# B&R Automation Studio project CControl (part 3)

#### Main.st
```iecst
PROGRAM _INIT

END_PROGRAM

PROGRAM _CYCLIC

	//Zeitticks generieren
	fbLascoZdxx_0(IN 	:= Echtzeit.Sekunde);
	sekTick				:= fbLascoZdxx_0.Q;

	//Modul 2 bei Entfeuchter-Typen 7, 8, 9 und 10 (10 ist Reserve, eigene Einstellungen möglich)
	gModul2Vorhanden	:= (Betriebsparameter.Entfeuchter.IndexType = 7) OR (Betriebsparameter.Entfeuchter.IndexType = 8) OR (Betriebsparameter.Entfeuchter.IndexType = 9) OR
	(Betriebsparameter.Entfeuchter.IndexType = 10);

	//Ölsumpheizung Modul 1 **********************************************************************************************************************************************************************

	//Eingänge
	Aktoren.OelsumpfheizungModul1.EintrittTemp					:= aiEintrittTemperatur;
	Aktoren.OelsumpfheizungModul1.StatusSensorEintrittOk		:= NOT alarmFehler[FEHLER_SENSOR_EINTRITT];

	//GUI-Parameter
	Aktoren.OelsumpfheizungModul1.parTempOelsumpfheizungEin		:= 0.0;
	Aktoren.OelsumpfheizungModul1.parTempOelsumpfheizungAus		:= 0.0;

	//Ausgänge
	doOelsumpfheizungEinModul1									:= Aktoren.OelsumpfheizungModul1.OelsumpfheizungEin;

	//Status
	IF  doOelsumpfheizungEinModul1 THEN
		gStatusAnlage.Aktor[AKTOR_OELSUMPFHEIZUNG_MOD1]	:= STATUS_AKTIV;
	ELSE
		gStatusAnlage.Aktor[AKTOR_OELSUMPFHEIZUNG_MOD1]	:= STATUS_NICHT_AKTIV;
	END_IF

	//Ölsumpheizung Modul 2 **********************************************************************************************************************************************************************

	//Eingänge
	Aktoren.OelsumpfheizungModul2.EintrittTemp					:= aiEintrittTemperatur;
	Aktoren.OelsumpfheizungModul2.StatusSensorEintrittOk		:= NOT alarmFehler[FEHLER_SENSOR_EINTRITT];

	//GUI-Parameter
	Aktoren.OelsumpfheizungModul2.parTempOelsumpfheizungEin		:= 0.0;
	Aktoren.OelsumpfheizungModul2.parTempOelsumpfheizungAus		:= 0.0;

	//Ausgänge
	doOelsumpfheizungEinModul2										:= Aktoren.OelsumpfheizungModul2.OelsumpfheizungEin;

	//Status
	IF  doOelsumpfheizungEinModul2 THEN
		gStatusAnlage.Aktor[AKTOR_OELSUMPFHEIZUNG_MOD2]	:= STATUS_AKTIV;
	ELSE
		gStatusAnlage.Aktor[AKTOR_OELSUMPFHEIZUNG_MOD2]	:= STATUS_NICHT_AKTIV;
	END_IF

	//Kompressor Modul 1 **********************************************************************************************************************************************************************

	//Eingänge
	Aktoren.KompressorModul1.EintrittFeuchte			:= aiEintrittFeuchte;
	Aktoren.KompressorModul1.Niederdruck				:= aiNiederdruckModul1;
	Aktoren.KompressorModul1.Hochdruck					:= aiHochdruckModul1;
	Aktoren.KompressorModul1.KlappenumschaltungAkiv		:= Aktoren.VentUndKlappen.UmschaltungAktiv OR Strombegrenzung.StrombegrenzungEin OR
	(diDrehzahlbegrVentilator1 AND Boxen.EntfeuchterVonVent1Abhaengig) OR (diDrehzahlbegrVentilator2 AND Boxen.EntfeuchterVonVent2Abhaengig);
	Aktoren.KompressorModul1.BetriebsmldgVentilator		:= (doVentilator1Ein AND Boxen.EntfeuchterVonVent1Abhaengig) OR
	(doVentilator2Ein AND Boxen.EntfeuchterVonVent2Abhaengig) OR (diVentilator1InBetrieb AND Boxen.EntfeuchterInselbetrieb);
	Aktoren.KompressorModul1.BetriebsmldgKompressor		:= diBetriebsmldgKompressorModul1;
	Aktoren.KompressorModul1.StatusSensorEintrittOk		:= NOT alarmFehler[FEHLER_SENSOR_EINTRITT];
	Aktoren.KompressorModul1.StatusSensorNiederdruckOk	:= NOT alarmFehler[FEHLER_SENSOR_NIEDERDRUCK_MOD1];
	Aktoren.KompressorModul1.diHochdruckOk				:= diHochdruckOkModul1;
	Aktoren.KompressorModul1.diNiederdruckOk			:= diNiederdruckOkModul1;
	Aktoren.KompressorModul1.SicherheitOk				:= NOT alarmFehler[FEHLER_HOCHDRUCK_MODUL1] AND NOT alarmFehler[FEHLER_NIEDERDRUCK_MODUL1] AND NOT alarmFehler[FEHLER_VOLLSCHUTZ_KOMPR_MOD1] AND NOT
	alarmFehler[FEHLER_OELDRUCK_KOMPR_MOD1] AND NOT alarmFehler[FEHLER_EINTRITT_TEMP_ZU_HOCH] AND NOT alarmFehler[FEHLER_EINTRITT_TEMP_ZU_NIEDRIG];

	//GUI-Parameter
	Aktoren.KompressorModul1.QuitFehler						:= hmiButtons.QuitFehler;
	Aktoren.KompressorModul1.parEinschaltverzAbtau			:= Betriebsparameter.Entfeuchter.EinschaltverzAbtau;
	Aktoren.KompressorModul1.parAusschaltverzAbtau			:= Betriebsparameter.Entfeuchter.AusschaltverzAbtau;
	Aktoren.KompressorModul1.parEinschaltverzKompressor		:= Betriebsparameter.Entfeuchter.EinschaltverzKompressor;
	Aktoren.KompressorModul1.parEinschaltverzMagnetventil	:= Betriebsparameter.Kompressor1.EinschaltverzMagnetventil;
	Aktoren.KompressorModul1.parFeuchteEin					:= Betriebsparameter.Entfeuchter.EintrittFeuchteEin;
	Aktoren.KompressorModul1.parFeuchteAus					:= Betriebsparameter.Entfeuchter.EintrittFeuchteAus;
	Aktoren.KompressorModul1.parNiederdruckMin				:= Betriebsparameter.Kompressor1.NiederdruckMin;
	Aktoren.KompressorModul1.parNiederdruckMax				:= Betriebsparameter.Kompressor1.NiederdruckMax;
	Aktoren.KompressorModul1.parNiederdruckPumpdown			:= Betriebsparameter.Kompressor1.NiederdruckPumpDown;
	Aktoren.KompressorModul1.parHochdruckMax				:= Betriebsparameter.Kompressor1.HochdruckMax;
	Aktoren.KompressorModul1.parVerzStandbyBeiKlappenumsch	:= Betriebsparameter.Entfeuchter.VerzStandbyHochdruckMax;
	Aktoren.KompressorModul1.DrehzahlMin					:= Betriebsparameter.Kompressor1.DrehzahlMin;
	Aktoren.KompressorModul1.DrehzahlMax					:= Betriebsparameter.Kompressor1.DrehzahlMax;
	Aktoren.KompressorModul1.RampeUp						:= Betriebsparameter.Kompressor1.RampeUp;
	Aktoren.KompressorModul1.RampeDown						:= Betriebsparameter.Kompressor1.RampeDown;

	//Ausgänge
	doKompressorEinModul1									:= Aktoren.KompressorModul1.FreigabeKompressorOut AND diHochdruckOkModul1 AND diNiederdruckOkModul1;
	aoDrehzahlvorgKompressorModul1							:= Aktoren.KompressorModul1.DrehzahlOut;
	doMagnetventilEinModul1									:= Aktoren.KompressorModul1.MagnetventilOut;

	//Status
	IF doKompressorEinModul1 THEN
		gStatusAnlage.Aktor[AKTOR_KOMPRESSOR_MOD1]			:= STATUS_AKTIV;
	ELSIF Aktoren.KompressorModul1.StoerungOut THEN
		gStatusAnlage.Aktor[AKTOR_KOMPRESSOR_MOD1]			:= STATUS_STOERUNG;
	ELSIF (Aktoren.KompressorModul1.Automatik OR Aktoren.KompressorModul1.Dauerbetrieb) AND Boxen.FreigabeLuftentfeuchter AND NOT doKompressorEinModul1 THEN
		gStatusAnlage.Aktor[AKTOR_KOMPRESSOR_MOD1]			:= STATUS_ENTF_STANDBY;
	ELSIF Aktoren.KompressorModul1.AbtauungAktiv THEN
		gStatusAnlage.Aktor[AKTOR_KOMPRESSOR_MOD1]			:= STATUS_ENTF_ABTAUUNG;
	ELSE
		gStatusAnlage.Aktor[AKTOR_KOMPRESSOR_MOD1]			:= STATUS_NICHT_AKTIV;
	END_IF

	//Status
	IF  doMagnetventilEinModul1 THEN
		gStatusAnlage.Aktor[AKTOR_MAGNETVENTIL_MOD1]		:= STATUS_AKTIV;
	ELSE
		gStatusAnlage.Aktor[AKTOR_MAGNETVENTIL_MOD1]		:= STATUS_NICHT_AKTIV;
	END_IF

	//Kompressor Modul 2 **********************************************************************************************************************************************************************

	//Eingänge
	Aktoren.KompressorModul2.EintrittFeuchte			:= aiEintrittFeuchte;
	Aktoren.KompressorModul2.Niederdruck				:= aiNiederdruckModul2;
	Aktoren.KompressorModul2.Hochdruck					:= aiHochdruckModul2;
	Aktoren.KompressorModul2.KlappenumschaltungAkiv		:= Aktoren.VentUndKlappen.UmschaltungAktiv OR Strombegrenzung.StrombegrenzungEin OR
	(diDrehzahlbegrVentilator1 AND Boxen.EntfeuchterVonVent1Abhaengig) OR (diDrehzahlbegrVentilator2 AND Boxen.EntfeuchterVonVent2Abhaengig);
	Aktoren.KompressorModul2.BetriebsmldgVentilator		:= (doVentilator1Ein AND Boxen.EntfeuchterVonVent1Abhaengig) OR
	(doVentilator2Ein AND Boxen.EntfeuchterVonVent2Abhaengig) OR (diVentilator1InBetrieb AND Boxen.EntfeuchterInselbetrieb);
	Aktoren.KompressorModul2.BetriebsmldgKompressor		:= diBetriebsmldgKompressorModul2;
	Aktoren.KompressorModul2.StatusSensorEintrittOk		:= NOT alarmFehler[FEHLER_SENSOR_EINTRITT];
	Aktoren.KompressorModul2.StatusSensorNiederdruckOk	:= NOT alarmFehler[FEHLER_SENSOR_NIEDERDRUCK_MOD2];
	Aktoren.KompressorModul2.diHochdruckOk				:= diHochdruckOkModul2;
	Aktoren.KompressorModul2.diNiederdruckOk			:= diNiederdruckOkModul2;
	Aktoren.KompressorModul2.SicherheitOk				:= NOT alarmFehler[FEHLER_HOCHDRUCK_MODUL2] AND NOT alarmFehler[FEHLER_NIEDERDRUCK_MODUL2] AND NOT alarmFehler[FEHLER_VOLLSCHUTZ_KOMPR_MOD2] AND NOT
	alarmFehler[FEHLER_OELDRUCK_KOMPR_MOD2] AND NOT alarmFehler[FEHLER_EINTRITT_TEMP_ZU_HOCH] AND NOT alarmFehler[FEHLER_EINTRITT_TEMP_ZU_NIEDRIG];

	//GUI-Parameter
	Aktoren.KompressorModul2.QuitFehler						:= hmiButtons.QuitFehler;
	Aktoren.KompressorModul2.parEinschaltverzAbtau			:= Betriebsparameter.Entfeuchter.EinschaltverzAbtau;
	Aktoren.KompressorModul2.parAusschaltverzAbtau			:= Betriebsparameter.Entfeuchter.AusschaltverzAbtau;
	Aktoren.KompressorModul2.parEinschaltverzKompressor		:= Betriebsparameter.Entfeuchter.EinschaltverzKompressor + Betriebsparameter.Entfeuchter.AnlaufverzModul2;
	Aktoren.KompressorModul2.parEinschaltverzMagnetventil	:= Betriebsparameter.Kompressor1.EinschaltverzMagnetventil;
	Aktoren.KompressorModul2.parFeuchteEin					:= Betriebsparameter.Entfeuchter.EintrittFeuchteEin;
	Aktoren.KompressorModul2.parFeuchteAus					:= Betriebsparameter.Entfeuchter.EintrittFeuchteAus;
	Aktoren.KompressorModul2.parNiederdruckMin				:= Betriebsparameter.Kompressor1.NiederdruckMin;
	Aktoren.KompressorModul2.parNiederdruckMax				:= Betriebsparameter.Kompressor1.NiederdruckMax;
	Aktoren.KompressorModul2.parNiederdruckPumpdown			:= Betriebsparameter.Kompressor1.NiederdruckPumpDown;
	Aktoren.KompressorModul2.parHochdruckMax				:= Betriebsparameter.Kompressor1.HochdruckMax;
	Aktoren.KompressorModul2.parVerzStandbyBeiKlappenumsch	:= Betriebsparameter.Entfeuchter.VerzStandbyHochdruckMax;
	Aktoren.KompressorModul2.DrehzahlMin					:= Betriebsparameter.Kompressor2.DrehzahlMin;
	Aktoren.KompressorModul2.DrehzahlMax					:= Betriebsparameter.Kompressor2.DrehzahlMax;
	Aktoren.KompressorModul2.RampeUp						:= Betriebsparameter.Kompressor2.RampeUp;
	Aktoren.KompressorModul2.RampeDown						:= Betriebsparameter.Kompressor2.RampeDown;

	//Ausgänge
	doKompressorEinModul2									:= Aktoren.KompressorModul2.FreigabeKompressorOut AND diHochdruckOkModul2 AND diNiederdruckOkModul2;
	aoDrehzahlvorgKompressorModul2							:= Aktoren.KompressorModul2.DrehzahlOut;
	doMagnetventilEinModul2									:= Aktoren.KompressorModul2.MagnetventilOut;

	//Status
	IF doKompressorEinModul2 THEN
		gStatusAnlage.Aktor[AKTOR_KOMPRESSOR_MOD2]			:= STATUS_AKTIV;
	ELSIF Aktoren.KompressorModul2.StoerungOut THEN
		gStatusAnlage.Aktor[AKTOR_KOMPRESSOR_MOD2]			:= STATUS_STOERUNG;
	ELSIF (Aktoren.KompressorModul2.Automatik OR Aktoren.KompressorModul2.Dauerbetrieb) AND Boxen.FreigabeLuftentfeuchter AND NOT doKompressorEinModul2 THEN
		gStatusAnlage.Aktor[AKTOR_KOMPRESSOR_MOD2]			:= STATUS_ENTF_STANDBY;
	ELSIF Aktoren.KompressorModul2.AbtauungAktiv THEN
		gStatusAnlage.Aktor[AKTOR_KOMPRESSOR_MOD2]			:= STATUS_ENTF_ABTAUUNG;
	ELSE
		gStatusAnlage.Aktor[AKTOR_KOMPRESSOR_MOD2]			:= STATUS_NICHT_AKTIV;
	END_IF

	//Status
	IF  doMagnetventilEinModul2 THEN
		gStatusAnlage.Aktor[AKTOR_MAGNETVENTIL_MOD2]		:= STATUS_AKTIV;
	ELSE
		gStatusAnlage.Aktor[AKTOR_MAGNETVENTIL_MOD2]		:= STATUS_NICHT_AKTIV;
	END_IF

	//Entfeuchter Fremdgerät **********************************************************************************************************************************************************************

	//Eingänge
	Aktoren.EntfeuchterFremd.BetriebsmldgEntfeuchter	:= diEntfeuchterFremdInBetrieb;
	Aktoren.EntfeuchterFremd.BetriebsmldgVentilator		:= diVentilator1InBetrieb;

	Aktoren.EntfeuchterFremd.WitterungIstSchlecht		:= (fbSchlechtwetterBox1.WetterIstSchlecht AND Betriebsparameter.Boxen[1].Luftentfeuchter AND Boxen.Box1Out.BoxAktiv) OR
	(fbSchlechtwetterBox2.WetterIstSchlecht AND Betriebsparameter.Boxen[2].Luftentfeuchter AND Boxen.Box2Out.BoxAktiv) OR
	(fbSchlechtwetterBox3.WetterIstSchlecht AND Betriebsparameter.Boxen[3].Luftentfeuchter AND Boxen.Box3Out.BoxAktiv) OR
	(fbSchlechtwetterBox4.WetterIstSchlecht AND Betriebsparameter.Boxen[4].Luftentfeuchter AND Boxen.Box4Out.BoxAktiv) OR
	(fbSchlechtwetterBox5.WetterIstSchlecht AND Betriebsparameter.Boxen[5].Luftentfeuchter AND Boxen.Box5Out.BoxAktiv) OR
	(fbSchlechtwetterBox6.WetterIstSchlecht AND Betriebsparameter.Boxen[6].Luftentfeuchter AND Boxen.Box6Out.BoxAktiv);
	Aktoren.EntfeuchterFremd.StoerungIn					:= diEntfeuchterFremdStoerung;

	//GUI-Parameter
	Aktoren.EntfeuchterFremd.parEinschaltverzKompressor	:= Betriebsparameter.Entfeuchter.EinschaltverzKompressor;
	Aktoren.EntfeuchterFremd.parVerzBetriebEntfeuchter	:= Betriebsparameter.Entfeuchter.VerzBetriebsmeldung;
	Aktoren.EntfeuchterFremd.parVerzStoerung			:= REAL_TO_UDINT(Betriebsparameter.Allgemein.VerzoegerungFehler * 1000);
	Aktoren.EntfeuchterFremd.QuitFehler					:= hmiButtons.QuitFehler;

	//Ausgänge
	doEntfFremdFreigabe									:= Aktoren.EntfeuchterFremd.FreigabeKompressorOut;

	//Status
	IF doEntfFremdFreigabe THEN
		IF diEntfeuchterFremdInBetrieb THEN
			gStatusAnlage.Aktor[AKTOR_ENTFEUCHTER_FREMD]		:= STATUS_AKTIV;
		ELSE
			gStatusAnlage.Aktor[AKTOR_ENTFEUCHTER_FREMD]		:= STATUS_ENTF_STANDBY;
		END_IF
	ELSIF Aktoren.EntfeuchterFremd.StoerungOut THEN
		gStatusAnlage.Aktor[AKTOR_ENTFEUCHTER_FREMD]		:= STATUS_STOERUNG;
	ELSE
		gStatusAnlage.Aktor[AKTOR_ENTFEUCHTER_FREMD]		:= STATUS_NICHT_AKTIV;
	END_IF

	//Abluftklappe **********************************************************************************************************************************************************************

	//Eingänge
	Aktoren.Abluftklappe.AbluftFeuchteIst			:= aiAbluftFeuchte;
	Aktoren.Abluftklappe.EndlageOffen				:= diAbluftklappeOffen;
	Aktoren.Abluftklappe.EndlageGeschl				:= diAbluftklappeGeschl;

	//GUI-Parameter
	Aktoren.Abluftklappe.AbluftFeuchteSoll			:= Betriebsparameter.Abluftklappe.AbluftfeuchteMax;
	Aktoren.Abluftklappe.Hysterese					:= Betriebsparameter.Abluftklappe.Hysterese;
	Aktoren.Abluftklappe.Laufzeit					:= Betriebsparameter.Abluftklappe.Laufzeit;
	Aktoren.Abluftklappe.Quit						:= hmiButtons.QuitFehler;

	//Ausgänge
	doAbluftklappeFreigabe							:= Aktoren.Abluftklappe.OeffnenOut AND NOT Aktoren.Abluftklappe.SchliessenOut;
	doAbluftklappeOeffnen							:= Aktoren.Abluftklappe.OeffnenOut;
	doAbluftklappeSchliessen						:= Aktoren.Abluftklappe.SchliessenOut;

	//Status
	IF doAbluftklappeFreigabe AND NOT diAbluftklappeOffen AND (Betriebsparameter.Abluftklappe.Laufzeit <> 0) THEN
		gStatusAnlage.Aktor[AKTOR_ABLUFTKLAPPE]			:= STATUS_AKTIV;
	ELSIF (NOT doAbluftklappeFreigabe) AND NOT diAbluftklappeGeschl AND (Betriebsparameter.Abluftklappe.Laufzeit <> 0) THEN
		gStatusAnlage.Aktor[AKTOR_ABLUFTKLAPPE]			:= STATUS_AKTIV;
	ELSIF Aktoren.Abluftklappe.FehlerLaufzeit THEN
		gStatusAnlage.Aktor[AKTOR_ABLUFTKLAPPE]			:= STATUS_STOERUNG;
	ELSIF doAbluftklappeFreigabe AND (diAbluftklappeOffen OR (Betriebsparameter.Abluftklappe.Laufzeit = 0)) THEN
		gStatusAnlage.Aktor[AKTOR_ABLUFTKLAPPE]			:= STATUS_OFFEN;
	ELSIF (NOT doAbluftklappeFreigabe) AND (diAbluftklappeGeschl OR (Betriebsparameter.Abluftklappe.Laufzeit = 0)) THEN
		gStatusAnlage.Aktor[AKTOR_ABLUFTKLAPPE]			:= STATUS_GESCHLOSSEN;
	ELSE
		gStatusAnlage.Aktor[AKTOR_ABLUFTKLAPPE]			:= STATUS_NICHT_AKTIV;
	END_IF

	//Abluftventilator **********************************************************************************************************************************************************************

	//Eingänge
	Aktoren.Abluftventilator.AbluftFeuchteIst		:= aiAbluftFeuchte;
	Aktoren.Abluftventilator.VentilatorInBetrieb	:= diAbluftventInBetrieb;
	Aktoren.Abluftventilator.RampeUp				:= 10;
	Aktoren.Abluftventilator.RampeDown				:= 10;

	//GUI-Parameter
	Aktoren.Abluftventilator.DrehzahlMin			:= Betriebsparameter.Abluftventilator.DrehzahlMin;
	Aktoren.Abluftventilator.DrehzahlMax			:= Betriebsparameter.Abluftventilator.DrehzahlMax;
	Aktoren.Abluftventilator.AbluftFeuchteSoll		:= Betriebsparameter.Abluftventilator.AbluftfeuchteMax;
	Aktoren.Abluftventilator.Hysterese				:= Betriebsparameter.Abluftventilator.Hysterese;
	Aktoren.Abluftventilator.QuitFehler				:= hmiButtons.QuitFehler;

	//Ausgänge
	doAbluftventilatorEin							:= Aktoren.Abluftventilator.FreigabeVentilatorOut;
	aoDrehzahlvorgAbluftventilator					:= Aktoren.Abluftventilator.DrehzahlVentilatorOut;

	//Status
	IF doAbluftventilatorEin THEN
		gStatusAnlage.Aktor[AKTOR_ABLUFTVENTILATOR]		:= STATUS_AKTIV;
	ELSIF Aktoren.Abluftventilator.FehlerOut THEN
		gStatusAnlage.Aktor[AKTOR_ABLUFTVENTILATOR]		:= STATUS_STOERUNG;
	ELSE
		gStatusAnlage.Aktor[AKTOR_ABLUFTVENTILATOR]		:= STATUS_NICHT_AKTIV;
	END_IF

	//Ventilatoren, Bypassklappe, Umschaltklappen und Klappen für Boxen **********************************************************************************************************************

	//Eingänge
	Aktoren.VentUndKlappen.Freigabe						:= TRUE;
	Aktoren.VentUndKlappen.BypassklVonVent1Abhaengig	:= Boxen.BypassklVonVent1Abhaengig;
	Aktoren.VentUndKlappen.BypassklVonVent2Abhaengig	:= Boxen.BypassklVonVent2Abhaengig;
	Aktoren.VentUndKlappen.Boxenkl1VonVent1Abhaengig	:= Boxen.Boxenkl1VonVent1Abhaengig;
	Aktoren.VentUndKlappen.Boxenkl2VonVent1Abhaengig	:= Boxen.Boxenkl2VonVent1Abhaengig;
	Aktoren.VentUndKlappen.Boxenkl3VonVent1Abhaengig	:= Boxen.Boxenkl3VonVent1Abhaengig;
	Aktoren.VentUndKlappen.Boxenkl4VonVent1Abhaengig	:= Boxen.Boxenkl4VonVent1Abhaengig;
	Aktoren.VentUndKlappen.Boxenkl5VonVent1Abhaengig	:= Boxen.Boxenkl5VonVent1Abhaengig;
	Aktoren.VentUndKlappen.Boxenkl6VonVent1Abhaengig	:= Boxen.Boxenkl6VonVent1Abhaengig;
	Aktoren.VentUndKlappen.Boxenkl1VonVent2Abhaengig	:= Boxen.Boxenkl1VonVent2Abhaengig;
	Aktoren.VentUndKlappen.Boxenkl2VonVent2Abhaengig	:= Boxen.Boxenkl2VonVent2Abhaengig;
	Aktoren.VentUndKlappen.Boxenkl3VonVent2Abhaengig	:= Boxen.Boxenkl3VonVent2Abhaengig;
	Aktoren.VentUndKlappen.Boxenkl4VonVent2Abhaengig	:= Boxen.Boxenkl4VonVent2Abhaengig;
	Aktoren.VentUndKlappen.Boxenkl5VonVent2Abhaengig	:= Boxen.Boxenkl5VonVent2Abhaengig;
	Aktoren.VentUndKlappen.Boxenkl6VonVent2Abhaengig	:= Boxen.Boxenkl6VonVent2Abhaengig;
	Aktoren.VentUndKlappen.UmluftklVonVent1Abhaengig	:= Betriebsparameter.Ausstattung.Vent1AusWennUmschUmluftkl;
	Aktoren.VentUndKlappen.UmluftklVonVent2Abhaengig	:= Betriebsparameter.Ausstattung.Vent2AusWennUmschUmluftkl;
	Aktoren.VentUndKlappen.EndlBoxenklappe1Geschl		:= diBox1Geschl;
	Aktoren.VentUndKlappen.EndlBoxenklappe1Offen		:= diBox1Offen;
	Aktoren.VentUndKlappen.EndlBoxenklappe2Geschl		:= diBox2Geschl;
	Aktoren.VentUndKlappen.EndlBoxenklappe2Offen		:= diBox2Offen;
	Aktoren.VentUndKlappen.EndlBoxenklappe3Geschl		:= diBox3Geschl;
	Aktoren.VentUndKlappen.EndlBoxenklappe3Offen		:= diBox3Offen;
	Aktoren.VentUndKlappen.EndlBoxenklappe4Geschl		:= diBox4Geschl;
	Aktoren.VentUndKlappen.EndlBoxenklappe4Offen		:= diBox4Offen;
	Aktoren.VentUndKlappen.EndlBoxenklappe5Geschl		:= diBox5Geschl;
	Aktoren.VentUndKlappen.EndlBoxenklappe5Offen		:= diBox5Offen;
	Aktoren.VentUndKlappen.EndlBoxenklappe6Geschl		:= diBox6Geschl;
	Aktoren.VentUndKlappen.EndlBoxenklappe6Offen		:= diBox6Offen;
	Aktoren.VentUndKlappen.EndlBypassGeschl				:= diBypassklappeGeschl;
	Aktoren.VentUndKlappen.EndlBypassOffen				:= diBypassklappeOffen;
	Aktoren.VentUndKlappen.EndlBypassGeschl				:= diBypassklappeGeschl;
	Aktoren.VentUndKlappen.EndlBypassOffen				:= diBypassklappeOffen;
	Aktoren.VentUndKlappen.EndlUmschaltkl1Geschl		:= diUmschaltklappe1Geschl;
	Aktoren.VentUndKlappen.EndlUmschaltkl1Offen			:= diUmschaltklappe1Offen;
	Aktoren.VentUndKlappen.EndlUmschaltkl2Geschl		:= diUmschaltklappe2Geschl;
	Aktoren.VentUndKlappen.EndlUmschaltkl2Offen			:= diUmschaltklappe2Offen;
	Aktoren.VentUndKlappen.LuftaufbereitungInBetrieb	:= doKompressorEinModul1 OR doKompressorEinModul2 OR Aktoren.Warmluftofen.WarmluftofenAktiv OR
	Aktoren.Scheitholzofen.ScheitholzofenAktiv OR doHeizregisterEin;
	Aktoren.VentUndKlappen.Ventilator1InBetrieb			:= diVentilator1InBetrieb;
	Aktoren.VentUndKlappen.Ventilator2InBetrieb			:= diVentilator2InBetrieb;
	Aktoren.VentUndKlappen.Boxenklappe1Vorhanden		:= (Betriebsparameter.Boxen[1].StellungKlappe1 <> FBBOX_NICHT_VERWENDET) OR
	(Betriebsparameter.Boxen[2].StellungKlappe1 <> FBBOX_NICHT_VERWENDET) OR (Betriebsparameter.Boxen[3].StellungKlappe1 <> FBBOX_NICHT_VERWENDET) OR
	(Betriebsparameter.Boxen[4].StellungKlappe1 <> FBBOX_NICHT_VERWENDET) OR (Betriebsparameter.Boxen[5].StellungKlappe1 <> FBBOX_NICHT_VERWENDET) OR
	(Betriebsparameter.Boxen[6].StellungKlappe1 <> FBBOX_NICHT_VERWENDET);
	Aktoren.VentUndKlappen.Boxenklappe2Vorhanden		:= (Betriebsparameter.Boxen[1].StellungKlappe2 <> FBBOX_NICHT_VERWENDET) OR
	(Betriebsparameter.Boxen[2].StellungKlappe2 <> FBBOX_NICHT_VERWENDET) OR (Betriebsparameter.Boxen[3].StellungKlappe2 <> FBBOX_NICHT_VERWENDET) OR
	(Betriebsparameter.Boxen[4].StellungKlappe2 <> FBBOX_NICHT_VERWENDET) OR (Betriebsparameter.Boxen[5].StellungKlappe2 <> FBBOX_NICHT_VERWENDET) OR
	(Betriebsparameter.Boxen[6].StellungKlappe2 <> FBBOX_NICHT_VERWENDET);
	Aktoren.VentUndKlappen.Boxenklappe3Vorhanden		:= (Betriebsparameter.Boxen[1].StellungKlappe3 <> FBBOX_NICHT_VERWENDET) OR
	(Betriebsparameter.Boxen[2].StellungKlappe3 <> FBBOX_NICHT_VERWENDET) OR (Betriebsparameter.Boxen[3].StellungKlappe3 <> FBBOX_NICHT_VERWENDET) OR
	(Betriebsparameter.Boxen[4].StellungKlappe3 <> FBBOX_NICHT_VERWENDET) OR (Betriebsparameter.Boxen[5].StellungKlappe3 <> FBBOX_NICHT_VERWENDET) OR
	(Betriebsparameter.Boxen[6].StellungKlappe3 <> FBBOX_NICHT_VERWENDET);
	Aktoren.VentUndKlappen.Boxenklappe4Vorhanden		:= (Betriebsparameter.Boxen[1].StellungKlappe4 <> FBBOX_NICHT_VERWENDET) OR
	(Betriebsparameter.Boxen[2].StellungKlappe4 <> FBBOX_NICHT_VERWENDET) OR (Betriebsparameter.Boxen[3].StellungKlappe4 <> FBBOX_NICHT_VERWENDET) OR
	(Betriebsparameter.Boxen[4].StellungKlappe4 <> FBBOX_NICHT_VERWENDET) OR (Betriebsparameter.Boxen[5].StellungKlappe4 <> FBBOX_NICHT_VERWENDET) OR
	(Betriebsparameter.Boxen[6].StellungKlappe4 <> FBBOX_NICHT_VERWENDET);
	Aktoren.VentUndKlappen.Boxenklappe5Vorhanden		:= (Betriebsparameter.Boxen[1].StellungKlappe5 <> FBBOX_NICHT_VERWENDET) OR
	(Betriebsparameter.Boxen[2].StellungKlappe5 <> FBBOX_NICHT_VERWENDET) OR (Betriebsparameter.Boxen[3].StellungKlappe5 <> FBBOX_NICHT_VERWENDET) OR
	(Betriebsparameter.Boxen[4].StellungKlappe5 <> FBBOX_NICHT_VERWENDET) OR (Betriebsparameter.Boxen[5].StellungKlappe5 <> FBBOX_NICHT_VERWENDET) OR
	(Betriebsparameter.Boxen[6].StellungKlappe5 <> FBBOX_NICHT_VERWENDET);
	Aktoren.VentUndKlappen.Boxenklappe6Vorhanden		:= (Betriebsparameter.Boxen[1].StellungKlappe6 <> FBBOX_NICHT_VERWENDET) OR
	(Betriebsparameter.Boxen[2].StellungKlappe6 <> FBBOX_NICHT_VERWENDET) OR (Betriebsparameter.Boxen[3].StellungKlappe6 <> FBBOX_NICHT_VERWENDET) OR
	(Betriebsparameter.Boxen[4].StellungKlappe6 <> FBBOX_NICHT_VERWENDET) OR (Betriebsparameter.Boxen[5].StellungKlappe6 <> FBBOX_NICHT_VERWENDET) OR
	(Betriebsparameter.Boxen[6].StellungKlappe6 <> FBBOX_NICHT_VERWENDET);

	//GUI-Parameter
	Aktoren.VentUndKlappen.QuitFehler					:= hmiButtons.QuitFehler;
	Aktoren.VentUndKlappen.AnlaufverzZweiterVent		:= Betriebsparameter.Schrittkette.AnlaufverzZweiterVentilator;
	Aktoren.VentUndKlappen.DrehzahlVent1Min				:= Betriebsparameter.Ventilator1.DrehzahlMin;
	Aktoren.VentUndKlappen.DrehzahlVent1Max				:= Betriebsparameter.Ventilator1.DrehzahlMax;
	Aktoren.VentUndKlappen.RampeVent1Up					:= Betriebsparameter.Ventilator1.ZeitRampeUp;
	Aktoren.VentUndKlappen.RampeVent1Down				:= Betriebsparameter.Ventilator1.ZeitRampeDown;
	Aktoren.VentUndKlappen.DrehzahlVent1Umsch			:= Betriebsparameter.Ventilator1.DrzUmschaltung;
	Aktoren.VentUndKlappen.DrzVent1UmschMitLuftaufb		:= Betriebsparameter.Ventilator1.DrzUmschaltungMitLuftaufb;
	Aktoren.VentUndKlappen.DrehzahlVent2Min				:= Betriebsparameter.Ventilator2.DrehzahlMin;
	Aktoren.VentUndKlappen.DrehzahlVent2Max				:= Betriebsparameter.Ventilator2.DrehzahlMax;
	Aktoren.VentUndKlappen.RampeVent2Up					:= Betriebsparameter.Ventilator2.ZeitRampeUp;
	Aktoren.VentUndKlappen.RampeVent2Down				:= Betriebsparameter.Ventilator2.ZeitRampeDown;
	Aktoren.VentUndKlappen.DrehzahlVent2Umsch			:= Betriebsparameter.Ventilator2.DrzUmschaltung;
	Aktoren.VentUndKlappen.DrzVent2UmschMitLuftaufb		:= Betriebsparameter.Ventilator2.DrzUmschaltungMitLuftaufb;
	Aktoren.VentUndKlappen.LaufzeitBypassklappe			:= Betriebsparameter.Bypassklappe.Laufzeit;
	Aktoren.VentUndKlappen.LaufzeitBoxenklappe1			:= Betriebsparameter.KlappenBoxen[1].Laufzeit;
	Aktoren.VentUndKlappen.LaufzeitBoxenklappe2			:= Betriebsparameter.KlappenBoxen[2].Laufzeit;
	Aktoren.VentUndKlappen.LaufzeitBoxenklappe3			:= Betriebsparameter.KlappenBoxen[3].Laufzeit;
	Aktoren.VentUndKlappen.LaufzeitBoxenklappe4			:= Betriebsparameter.KlappenBoxen[4].Laufzeit;
	Aktoren.VentUndKlappen.LaufzeitBoxenklappe5			:= Betriebsparameter.KlappenBoxen[5].Laufzeit;
	Aktoren.VentUndKlappen.LaufzeitBoxenklappe6			:= Betriebsparameter.KlappenBoxen[6].Laufzeit;
	Aktoren.VentUndKlappen.LaufzeitUmschaltklappe1		:= Betriebsparameter.Umschaltklappen.LaufzeitKlappe1;
	Aktoren.VentUndKlappen.LaufzeitUmschaltklappe2		:= Betriebsparameter.Umschaltklappen.LaufzeitKlappe2;
	Aktoren.VentUndKlappen.EndlagenVhdBoxenklappe1		:= Betriebsparameter.Ausstattung.EndlagenVhdBoxenklappe1;
	Aktoren.VentUndKlappen.EndlagenVhdBoxenklappe2		:= Betriebsparameter.Ausstattung.EndlagenVhdBoxenklappe2;
	Aktoren.VentUndKlappen.EndlagenVhdBoxenklappe3		:= Betriebsparameter.Ausstattung.EndlagenVhdBoxenklappe3;
	Aktoren.VentUndKlappen.EndlagenVhdBoxenklappe4		:= Betriebsparameter.Ausstattung.EndlagenVhdBoxenklappe4;
	Aktoren.VentUndKlappen.EndlagenVhdBoxenklappe5		:= Betriebsparameter.Ausstattung.EndlagenVhdBoxenklappe5;
	Aktoren.VentUndKlappen.EndlagenVhdBoxenklappe6		:= Betriebsparameter.Ausstattung.EndlagenVhdBoxenklappe6;
	Aktoren.VentUndKlappen.EndlagenVhdUmschaltklappe1	:= Betriebsparameter.Ausstattung.EndlagenVhdUmschaltklappe1;
	Aktoren.VentUndKlappen.EndlagenVhdUmschaltklappe2	:= Betriebsparameter.Ausstattung.EndlagenVhdUmschaltklappe1;//Option Endlagen Umschaltklappen nur für beide Klappen gleich einstellbar
	Aktoren.VentUndKlappen.EndlagenVhdBypassklappe		:= Betriebsparameter.Ausstattung.EndlagenVhdBypassklappe;

	//Ausgänge
	doVentilator1Ein									:= Aktoren.VentUndKlappen.FreigabeVentilator1Out;
	doVentilator2Ein									:= Aktoren.VentUndKlappen.FreigabeVentilator2Out;
	aoDrehzahlvorgVentilator1							:= Aktoren.VentUndKlappen.DrehzahlVent1Out;
	aoDrehzahlvorgVentilator2							:= Aktoren.VentUndKlappen.DrehzahlVent2Out;
	doBypassklappeOeffnen								:= Aktoren.VentUndKlappen.BypassOeffnenOut;
	doBypassklappeSchliessen							:= Aktoren.VentUndKlappen.BypassSchliessenOut;
	doUmluftklappe1Freigabe								:= Aktoren.VentUndKlappen.Umschaltkl1OeffnenOut;
	doUmluftklappe1Oeffnen								:= Aktoren.VentUndKlappen.Umschaltkl1OeffnenOut;
	doUmluftklappe1Schliessen							:= Aktoren.VentUndKlappen.Umschaltkl1SchliessenOut;
	doUmluftklappe2Freigabe								:= Aktoren.VentUndKlappen.Umschaltkl2OeffnenOut;
	doUmluftklappe2Oeffnen								:= Aktoren.VentUndKlappen.Umschaltkl2OeffnenOut;
	doUmluftklappe2Schliessen							:= Aktoren.VentUndKlappen.Umschaltkl2SchliessenOut;
	doFreigabeBox1										:= Aktoren.VentUndKlappen.Boxenklappe1OeffnenOut;
	doFreigabeBox2										:= Aktoren.VentUndKlappen.Boxenklappe2OeffnenOut;
	doFreigabeBox3										:= Aktoren.VentUndKlappen.Boxenklappe3OeffnenOut;
	doFreigabeBox4										:= Aktoren.VentUndKlappen.Boxenklappe4OeffnenOut;
	doFreigabeBox5										:= Aktoren.VentUndKlappen.Boxenklappe5OeffnenOut;
	doFreigabeBox6										:= Aktoren.VentUndKlappen.Boxenklappe6OeffnenOut;

	//Status ***********************************************************************************************

	//Ventilator 1
	IF Aktoren.VentUndKlappen.FreigabeVentilator1Out THEN
		gStatusAnlage.Aktor[AKTOR_VENTILATOR_1]		:= STATUS_AKTIV;
	ELSIF Aktoren.VentUndKlappen.FehlerFuVentilator1 THEN
		gStatusAnlage.Aktor[AKTOR_VENTILATOR_1]		:= STATUS_STOERUNG;
	ELSE
		gStatusAnlage.Aktor[AKTOR_VENTILATOR_1]		:= STATUS_NICHT_AKTIV;
	END_IF

	//Ventilator 2
	IF Aktoren.VentUndKlappen.FreigabeVentilator2Out THEN
		gStatusAnlage.Aktor[AKTOR_VENTILATOR_2]		:= STATUS_AKTIV;
	ELSIF Aktoren.VentUndKlappen.FehlerFuVentilator2 THEN
		gStatusAnlage.Aktor[AKTOR_VENTILATOR_2]		:= STATUS_STOERUNG;
	ELSE
		gStatusAnlage.Aktor[AKTOR_VENTILATOR_2]		:= STATUS_NICHT_AKTIV;
	END_IF

	//Bypassklappe
	IF doBypassklappeOeffnen AND NOT (diBypassklappeOffen OR Aktoren.VentUndKlappen.BypassklappeIstOffen) AND (Betriebsparameter.Bypassklappe.Laufzeit <> 0) THEN
		gStatusAnlage.Aktor[AKTOR_BYPASSKLAPPE]	:= STATUS_AKTIV;
	ELSIF (NOT doBypassklappeOeffnen) AND NOT (diBypassklappeGeschl OR Aktoren.VentUndKlappen.BypassklappeIstGeschl) AND (Betriebsparameter.Bypassklappe.Laufzeit <> 0) THEN
		gStatusAnlage.Aktor[AKTOR_BYPASSKLAPPE]	:= STATUS_AKTIV;
	ELSIF doBypassklappeOeffnen AND ((diBypassklappeOffen OR Aktoren.VentUndKlappen.BypassklappeIstOffen) OR (Betriebsparameter.Bypassklappe.Laufzeit = 0)) THEN
		gStatusAnlage.Aktor[AKTOR_BYPASSKLAPPE]	:= STATUS_OFFEN;
	ELSIF (NOT doBypassklappeOeffnen) AND ((diBypassklappeGeschl OR Aktoren.VentUndKlappen.BypassklappeIstGeschl) OR (Betriebsparameter.Bypassklappe.Laufzeit = 0)) THEN
		gStatusAnlage.Aktor[AKTOR_BYPASSKLAPPE]	:= STATUS_GESCHLOSSEN;
	ELSIF Aktoren.VentUndKlappen.FehlerLaufzeitBypass THEN
		gStatusAnlage.Aktor[AKTOR_BYPASSKLAPPE]	:= STATUS_STOERUNG;
	ELSE
		gStatusAnlage.Aktor[AKTOR_BYPASSKLAPPE]	:= STATUS_NICHT_AKTIV;
	END_IF

	//Umluftklappe 1
	IF doUmluftklappe1Freigabe AND NOT (diUmschaltklappe1Offen OR Aktoren.VentUndKlappen.Umschaltklappe1IstOffen) AND (Betriebsparameter.Umschaltklappen.LaufzeitKlappe1 <> 0) AND Betriebsparameter.Ausstattung.Umschaltklappe1 THEN
		gStatusAnlage.Aktor[AKTOR_UMSCHALTKLAPPE_1]	:= STATUS_AKTIV;
	ELSIF (NOT doUmluftklappe1Freigabe) AND NOT (diUmschaltklappe1Geschl OR Aktoren.VentUndKlappen.Umschaltklappe1IstGeschl) AND (Betriebsparameter.Umschaltklappen.LaufzeitKlappe1 <> 0) AND Betriebsparameter.Ausstattung.Umschaltklappe1 THEN
		gStatusAnlage.Aktor[AKTOR_UMSCHALTKLAPPE_1]	:= STATUS_AKTIV;
	ELSIF doUmluftklappe1Freigabe AND ((diUmschaltklappe1Offen OR Aktoren.VentUndKlappen.Umschaltklappe1IstOffen) OR (Betriebsparameter.Umschaltklappen.LaufzeitKlappe1 = 0)) AND Betriebsparameter.Ausstattung.Umschaltklappe1 THEN
		gStatusAnlage.Aktor[AKTOR_UMSCHALTKLAPPE_1]	:= STATUS_OFFEN;
	ELSIF (NOT doUmluftklappe1Freigabe) AND ((diUmschaltklappe1Geschl OR Aktoren.VentUndKlappen.Umschaltklappe1IstGeschl) OR (Betriebsparameter.Umschaltklappen.LaufzeitKlappe1 = 0)) AND Betriebsparameter.Ausstattung.Umschaltklappe1 THEN
		gStatusAnlage.Aktor[AKTOR_UMSCHALTKLAPPE_1]	:= STATUS_GESCHLOSSEN;
	ELSIF Aktoren.VentUndKlappen.FehlerLaufzeitUmschaltkl1 AND Betriebsparameter.Ausstattung.Umschaltklappe1 THEN
		gStatusAnlage.Aktor[AKTOR_UMSCHALTKLAPPE_1]	:= STATUS_STOERUNG;
	ELSE
		gStatusAnlage.Aktor[AKTOR_UMSCHALTKLAPPE_1]	:= STATUS_NICHT_AKTIV;
	END_IF

	//Umluftklappe 2
	IF doUmluftklappe2Freigabe AND NOT (diUmschaltklappe2Offen OR Aktoren.VentUndKlappen.Umschaltklappe2IstOffen) AND (Betriebsparameter.Umschaltklappen.LaufzeitKlappe2 <> 0) AND Betriebsparameter.Ausstattung.Umschaltklappe2 THEN
		gStatusAnlage.Aktor[AKTOR_UMSCHALTKLAPPE_2]	:= STATUS_AKTIV;
	ELSIF (NOT doUmluftklappe2Freigabe) AND NOT (diUmschaltklappe2Geschl OR Aktoren.VentUndKlappen.Umschaltklappe2IstGeschl) AND (Betriebsparameter.Umschaltklappen.LaufzeitKlappe2 <> 0) AND Betriebsparameter.Ausstattung.Umschaltklappe2 THEN
		gStatusAnlage.Aktor[AKTOR_UMSCHALTKLAPPE_2]	:= STATUS_AKTIV;
	ELSIF doUmluftklappe2Freigabe AND ((diUmschaltklappe2Offen OR Aktoren.VentUndKlappen.Umschaltklappe2IstOffen) OR (Betriebsparameter.Umschaltklappen.LaufzeitKlappe2 = 0)) AND Betriebsparameter.Ausstattung.Umschaltklappe2 THEN
		gStatusAnlage.Aktor[AKTOR_UMSCHALTKLAPPE_2]	:= STATUS_OFFEN;
	ELSIF (NOT doUmluftklappe2Freigabe) AND ((diUmschaltklappe2Geschl OR Aktoren.VentUndKlappen.Umschaltklappe2IstGeschl) OR (Betriebsparameter.Umschaltklappen.LaufzeitKlappe2 = 0)) AND Betriebsparameter.Ausstattung.Umschaltklappe2 THEN
		gStatusAnlage.Aktor[AKTOR_UMSCHALTKLAPPE_2]	:= STATUS_GESCHLOSSEN;
	ELSIF Aktoren.VentUndKlappen.FehlerLaufzeitUmschaltkl2 AND Betriebsparameter.Ausstattung.Umschaltklappe2 THEN
		gStatusAnlage.Aktor[AKTOR_UMSCHALTKLAPPE_2]	:= STATUS_STOERUNG;
	ELSE
		gStatusAnlage.Aktor[AKTOR_UMSCHALTKLAPPE_2]	:= STATUS_NICHT_AKTIV;
	END_IF

	//Boxenklappe 1
	IF doFreigabeBox1 AND NOT (diBox1Offen OR Aktoren.VentUndKlappen.Boxenklappe1IstOffen) AND (Betriebsparameter.KlappenBoxen[1].Laufzeit <> 0) THEN
		gStatusAnlage.Aktor[AKTOR_KLAPPE_BOX_1]	:= STATUS_AKTIV;
	ELSIF (NOT doFreigabeBox1) AND NOT (diBox1Geschl OR Aktoren.VentUndKlappen.Boxenklappe1IstGeschl) AND (Betriebsparameter.KlappenBoxen[1].Laufzeit <> 0) THEN
		gStatusAnlage.Aktor[AKTOR_KLAPPE_BOX_1]	:= STATUS_AKTIV;
	ELSIF doFreigabeBox1 AND ((diBox1Offen OR Aktoren.VentUndKlappen.Boxenklappe1IstOffen) OR (Betriebsparameter.KlappenBoxen[1].Laufzeit = 0)) THEN
		gStatusAnlage.Aktor[AKTOR_KLAPPE_BOX_1]	:= STATUS_OFFEN;
	ELSIF (NOT doFreigabeBox1) AND ((diBox1Geschl OR Aktoren.VentUndKlappen.Boxenklappe1IstGeschl) OR (Betriebsparameter.KlappenBoxen[1].Laufzeit = 0)) THEN
		gStatusAnlage.Aktor[AKTOR_KLAPPE_BOX_1]	:= STATUS_GESCHLOSSEN;
	ELSIF Aktoren.VentUndKlappen.FehlerLaufzeitKlappeBox1 THEN
		gStatusAnlage.Aktor[AKTOR_KLAPPE_BOX_1]	:= STATUS_STOERUNG;
	ELSE
		gStatusAnlage.Aktor[AKTOR_KLAPPE_BOX_1]	:= STATUS_NICHT_AKTIV;
	END_IF

	//Boxenklappe 2
	IF doFreigabeBox2 AND NOT (diBox2Offen OR Aktoren.VentUndKlappen.Boxenklappe2IstOffen) AND (Betriebsparameter.KlappenBoxen[2].Laufzeit <> 0) THEN
		gStatusAnlage.Aktor[AKTOR_KLAPPE_BOX_2]	:= STATUS_AKTIV;
	ELSIF (NOT doFreigabeBox2) AND NOT (diBox2Geschl OR Aktoren.VentUndKlappen.Boxenklappe2IstGeschl) AND (Betriebsparameter.KlappenBoxen[2].Laufzeit <> 0) THEN
		gStatusAnlage.Aktor[AKTOR_KLAPPE_BOX_2]	:= STATUS_AKTIV;
	ELSIF doFreigabeBox2 AND ((diBox2Offen OR Aktoren.VentUndKlappen.Boxenklappe2IstOffen) OR (Betriebsparameter.KlappenBoxen[2].Laufzeit = 0)) THEN
		gStatusAnlage.Aktor[AKTOR_KLAPPE_BOX_2]	:= STATUS_OFFEN;
	ELSIF (NOT doFreigabeBox2) AND ((diBox2Geschl OR Aktoren.VentUndKlappen.Boxenklappe2IstGeschl) OR (Betriebsparameter.KlappenBoxen[2].Laufzeit = 0)) THEN
		gStatusAnlage.Aktor[AKTOR_KLAPPE_BOX_2]	:= STATUS_GESCHLOSSEN;
	ELSIF Aktoren.VentUndKlappen.FehlerLaufzeitKlappeBox2 THEN
		gStatusAnlage.Aktor[AKTOR_KLAPPE_BOX_2]	:= STATUS_STOERUNG;
	ELSE
		gStatusAnlage.Aktor[AKTOR_KLAPPE_BOX_2]	:= STATUS_NICHT_AKTIV;
	END_IF

	//Boxenklappe 3
	IF doFreigabeBox3 AND NOT (diBox3Offen OR Aktoren.VentUndKlappen.Boxenklappe3IstOffen) AND (Betriebsparameter.KlappenBoxen[3].Laufzeit <> 0) THEN
		gStatusAnlage.Aktor[AKTOR_KLAPPE_BOX_3]	:= STATUS_AKTIV;
	ELSIF (NOT doFreigabeBox3) AND NOT (diBox3Geschl OR Aktoren.VentUndKlappen.Boxenklappe3IstGeschl) AND (Betriebsparameter.KlappenBoxen[3].Laufzeit <> 0) THEN
		gStatusAnlage.Aktor[AKTOR_KLAPPE_BOX_3]	:= STATUS_AKTIV;
	ELSIF doFreigabeBox3 AND ((diBox3Offen OR Aktoren.VentUndKlappen.Boxenklappe3IstOffen) OR (Betriebsparameter.KlappenBoxen[3].Laufzeit = 0)) THEN
		gStatusAnlage.Aktor[AKTOR_KLAPPE_BOX_3]	:= STATUS_OFFEN;
	ELSIF (NOT doFreigabeBox3) AND ((diBox3Geschl OR Aktoren.VentUndKlappen.Boxenklappe3IstGeschl) OR (Betriebsparameter.KlappenBoxen[3].Laufzeit = 0)) THEN
		gStatusAnlage.Aktor[AKTOR_KLAPPE_BOX_3]	:= STATUS_GESCHLOSSEN;
	ELSIF Aktoren.VentUndKlappen.FehlerLaufzeitKlappeBox3 THEN
		gStatusAnlage.Aktor[AKTOR_KLAPPE_BOX_3]	:= STATUS_STOERUNG;
	ELSE
		gStatusAnlage.Aktor[AKTOR_KLAPPE_BOX_3]	:= STATUS_NICHT_AKTIV;
	END_IF

	//Boxenklappe 4
	IF doFreigabeBox4 AND NOT (diBox4Offen OR Aktoren.VentUndKlappen.Boxenklappe4IstOffen) AND (Betriebsparameter.KlappenBoxen[4].Laufzeit <> 0) THEN
		gStatusAnlage.Aktor[AKTOR_KLAPPE_BOX_4]	:= STATUS_AKTIV;
	ELSIF (NOT doFreigabeBox4) AND NOT (diBox4Geschl OR Aktoren.VentUndKlappen.Boxenklappe4IstGeschl) AND (Betriebsparameter.KlappenBoxen[4].Laufzeit <> 0) THEN
		gStatusAnlage.Aktor[AKTOR_KLAPPE_BOX_4]	:= STATUS_AKTIV;
	ELSIF doFreigabeBox4 AND ((diBox4Offen OR Aktoren.VentUndKlappen.Boxenklappe4IstOffen) OR (Betriebsparameter.KlappenBoxen[4].Laufzeit = 0)) THEN
		gStatusAnlage.Aktor[AKTOR_KLAPPE_BOX_4]	:= STATUS_OFFEN;
	ELSIF (NOT doFreigabeBox4) AND ((diBox4Geschl OR Aktoren.VentUndKlappen.Boxenklappe4IstGeschl) OR (Betriebsparameter.KlappenBoxen[4].Laufzeit = 0)) THEN
		gStatusAnlage.Aktor[AKTOR_KLAPPE_BOX_4]	:= STATUS_GESCHLOSSEN;
	ELSIF Aktoren.VentUndKlappen.FehlerLaufzeitKlappeBox4 THEN
		gStatusAnlage.Aktor[AKTOR_KLAPPE_BOX_4]	:= STATUS_STOERUNG;
	ELSE
		gStatusAnlage.Aktor[AKTOR_KLAPPE_BOX_4]	:= STATUS_NICHT_AKTIV;
	END_IF

	//Boxenklappe 5
	IF doFreigabeBox5 AND NOT (diBox5Offen OR Aktoren.VentUndKlappen.Boxenklappe5IstOffen) AND (Betriebsparameter.KlappenBoxen[5].Laufzeit <> 0) THEN
		gStatusAnlage.Aktor[AKTOR_KLAPPE_BOX_5]	:= STATUS_AKTIV;
	ELSIF (NOT doFreigabeBox5) AND NOT (diBox5Geschl OR Aktoren.VentUndKlappen.Boxenklappe5IstGeschl) AND (Betriebsparameter.KlappenBoxen[5].Laufzeit <> 0) THEN
		gStatusAnlage.Aktor[AKTOR_KLAPPE_BOX_5]	:= STATUS_AKTIV;
	ELSIF doFreigabeBox5 AND ((diBox5Offen OR Aktoren.VentUndKlappen.Boxenklappe5IstOffen) OR (Betriebsparameter.KlappenBoxen[5].Laufzeit = 0)) THEN
		gStatusAnlage.Aktor[AKTOR_KLAPPE_BOX_5]	:= STATUS_OFFEN;
	ELSIF (NOT doFreigabeBox5) AND ((diBox5Geschl OR Aktoren.VentUndKlappen.Boxenklappe5IstGeschl) OR (Betriebsparameter.KlappenBoxen[5].Laufzeit = 0)) THEN
		gStatusAnlage.Aktor[AKTOR_KLAPPE_BOX_5]	:= STATUS_GESCHLOSSEN;
	ELSIF Aktoren.VentUndKlappen.FehlerLaufzeitKlappeBox5 THEN
		gStatusAnlage.Aktor[AKTOR_KLAPPE_BOX_5]	:= STATUS_STOERUNG;
	ELSE
		gStatusAnlage.Aktor[AKTOR_KLAPPE_BOX_5]	:= STATUS_NICHT_AKTIV;
	END_IF

	//Boxenklappe 6
	IF doFreigabeBox6 AND NOT (diBox6Offen OR Aktoren.VentUndKlappen.Boxenklappe6IstOffen) AND (Betriebsparameter.KlappenBoxen[6].Laufzeit <> 0) THEN
		gStatusAnlage.Aktor[AKTOR_KLAPPE_BOX_6]	:= STATUS_AKTIV;
	ELSIF (NOT doFreigabeBox6) AND NOT (diBox6Geschl OR Aktoren.VentUndKlappen.Boxenklappe6IstGeschl) AND (Betriebsparameter.KlappenBoxen[6].Laufzeit <> 0) THEN
		gStatusAnlage.Aktor[AKTOR_KLAPPE_BOX_6]	:= STATUS_AKTIV;
	ELSIF doFreigabeBox6 AND ((diBox6Offen OR Aktoren.VentUndKlappen.Boxenklappe6IstOffen) OR (Betriebsparameter.KlappenBoxen[6].Laufzeit = 0)) THEN
		gStatusAnlage.Aktor[AKTOR_KLAPPE_BOX_6]	:= STATUS_OFFEN;
	ELSIF (NOT doFreigabeBox6) AND ((diBox6Geschl OR Aktoren.VentUndKlappen.Boxenklappe6IstGeschl) OR (Betriebsparameter.KlappenBoxen[6].Laufzeit = 0)) THEN
		gStatusAnlage.Aktor[AKTOR_KLAPPE_BOX_6]	:= STATUS_GESCHLOSSEN;
	ELSIF Aktoren.VentUndKlappen.FehlerLaufzeitKlappeBox6 THEN
		gStatusAnlage.Aktor[AKTOR_KLAPPE_BOX_6]	:= STATUS_STOERUNG;
	ELSE
		gStatusAnlage.Aktor[AKTOR_KLAPPE_BOX_6]	:= STATUS_NICHT_AKTIV;
	END_IF

	//Warmluftofen **********************************************************************************************************************************************************************
	//Steuerungsvariante <> HB4000/HB3000
	IF (hmiStatus.NameSteuerung <> 4) AND (hmiStatus.NameSteuerung <> 5) THEN

		//Eingänge
		Aktoren.Warmluftofen.BetriebsmeldungWarmluftofen	:= diWarmluftofenInBetrieb;
		Aktoren.Warmluftofen.FehlerSensorAussenluft			:= alarmFehler[FEHLER_SENSOR_FRISCHLUFT];
		Aktoren.Warmluftofen.FrischluftSattDefizitIst		:= gStatusAnlage.Berechnungen.FrischluftSattDefizit;

		//GUI-Parameter
		Aktoren.Warmluftofen.Auskuehlzeit					:= Betriebsparameter.Warmluftofen.Auskuehlzeit;
		Aktoren.Warmluftofen.FrischluftSattDefizitSoll		:= Betriebsparameter.Warmluftofen.SaettigungFrischlEin;
		Aktoren.Warmluftofen.Hysterese						:= Betriebsparameter.Warmluftofen.Hysterese;
		Aktoren.Warmluftofen.OptionBetriebsmldgVhd			:= Betriebsparameter.Ausstattung.WarmluftofenBetriebsmldg;
		Aktoren.Warmluftofen.QuitFehler						:= hmiButtons.QuitFehler;
		Aktoren.Warmluftofen.UmschaltverzWitterung			:= Betriebsparameter.Warmluftofen.VerzWetterwechsel;
		Aktoren.Warmluftofen.VerzBetriebsmeldung			:= Betriebsparameter.Warmluftofen.VerzBetriebsmeldung;
		Aktoren.Warmluftofen.WarmlufttemperaturVorgabe		:= Betriebsparameter.Warmluftofen.WarmlufttempVorgabeSoll;

	//HB4000/HB3000
	ELSE

		//Eingänge
		Aktoren.Warmluftofen.BetriebsmeldungWarmluftofen	:= diWarmluftofenInBetrieb;
		Aktoren.Warmluftofen.FehlerSensorAussenluft			:= FALSE;
		Aktoren.Warmluftofen.WetterIstSchlecht				:= gStatusAnlage.WetterIstSchlecht;

		//GUI-Parameter
		Aktoren.Warmluftofen.Auskuehlzeit					:= Betriebsparameter.Warmluftofen.Auskuehlzeit;
		Aktoren.Warmluftofen.OptionBetriebsmldgVhd			:= Betriebsparameter.Ausstattung.WarmluftofenBetriebsmldg;
		Aktoren.Warmluftofen.QuitFehler						:= hmiButtons.QuitFehler;
		Aktoren.Warmluftofen.VerzBetriebsmeldung			:= Betriebsparameter.Warmluftofen.VerzBetriebsmeldung;

	END_IF

	//Ausgänge
	doWarmluftofenEin									:= Aktoren.Warmluftofen.FreigabeWarmluftofenOut;
	aoTemperaturvorgWarmluftofen						:= Aktoren.Warmluftofen.WarmlufttempSollOut;

	//Status
	IF doWarmluftofenEin THEN
		gStatusAnlage.Aktor[AKTOR_WARMLUFTOFEN]		:= STATUS_AKTIV;
	ELSIF Aktoren.Warmluftofen.WarmluftofenAktiv THEN
		gStatusAnlage.Aktor[AKTOR_WARMLUFTOFEN]		:= STATUS_AUSKUEHLPHASE;
	ELSIF Aktoren.Warmluftofen.FehlerBetriebsmeldungOut OR Aktoren.Warmluftofen.FehlerSensorAussenluftOut THEN
		gStatusAnlage.Aktor[AKTOR_WARMLUFTOFEN]		:= STATUS_STOERUNG;
	ELSE
		gStatusAnlage.Aktor[AKTOR_WARMLUFTOFEN]		:= STATUS_NICHT_AKTIV;
	END_IF

	//Heizregister **********************************************************************************************************************************************************************
	//Steuerungsvariante <> HB4000/HB3000
	IF (hmiStatus.NameSteuerung <> 4) AND (hmiStatus.NameSteuerung <> 5) THEN

		//Eingänge
		Aktoren.Heizregister.FehlerSensorAussenluft			:= alarmFehler[FEHLER_SENSOR_FRISCHLUFT];
		Aktoren.Heizregister.FrischluftSattDefizitIst		:= gStatusAnlage.Berechnungen.FrischluftSattDefizit;

		//GUI-Parameter
		Aktoren.Heizregister.DrehzahlHeizregisterSoll		:= gCmdAnlage.Leistung.DrehzahlHeizregister;
		Aktoren.Heizregister.FrischluftSattDefizitSoll		:= Betriebsparameter.Heizregister.SaettigungFrischlEin;
		Aktoren.Heizregister.Hysterese						:= Betriebsparameter.Heizregister.Hysterese;
		Aktoren.Heizregister.QuitFehler						:= hmiButtons.QuitFehler;
		Aktoren.Heizregister.UmschaltverzWitterung			:= Betriebsparameter.Heizregister.VerzWetterwechsel;

		//Ausgänge
		doHeizregisterEin									:= Aktoren.Heizregister.FreigabeHeizregisterOut;
		aoLeistungsvorgHeizregister							:= Aktoren.Heizregister.DrehzahlHeizregisterOut;

		//HB4000/HB3000
	ELSE
		//Eingänge
		Aktoren.Heizregister.FehlerSensorAussenluft			:= FALSE;
		Aktoren.Heizregister.WetterIstSchlecht				:= gStatusAnlage.WetterIstSchlecht;

		//GUI-Parameter
		Aktoren.Heizregister.QuitFehler						:= hmiButtons.QuitFehler;

		//Ausgänge
		doHeizregisterEin									:= Aktoren.Heizregister.FreigabeHeizregisterOut;
	END_IF

	//Status
	IF doHeizregisterEin THEN
		gStatusAnlage.Aktor[AKTOR_HEIZREGISTER]		:= STATUS_AKTIV;
	ELSIF Aktoren.Heizregister.FehlerOut THEN
		gStatusAnlage.Aktor[AKTOR_HEIZREGISTER]		:= STATUS_STOERUNG;
	ELSE
		gStatusAnlage.Aktor[AKTOR_HEIZREGISTER]		:= STATUS_NICHT_AKTIV;
	END_IF

	//Scheitholzofen **********************************************************************************************************************************************************************

	//Eingänge
	Aktoren.Scheitholzofen.Betriebsmeldung		:= diScheitholzofenInBetrieb;

	//GUI-Parameter
	Aktoren.Scheitholzofen.Freigabe				:= Betriebsparameter.Ausstattung.Scheitholzofen;
	Aktoren.Scheitholzofen.Auskuehlzeit			:= Betriebsparameter.Scheitholzofen.Auskuehlzeit;

	//Ausgänge

	//Status
	IF diScheitholzofenInBetrieb THEN
		gStatusAnlage.Aktor[AKTOR_SCHEITHOLZOFEN]	:= STATUS_AKTIV;
	ELSIF Aktoren.Scheitholzofen.ScheitholzofenAktiv THEN
		gStatusAnlage.Aktor[AKTOR_SCHEITHOLZOFEN]	:= STATUS_AUSKUEHLPHASE;
	ELSE
		gStatusAnlage.Aktor[AKTOR_SCHEITHOLZOFEN]	:= STATUS_NICHT_AKTIV;
	END_IF

	//Notstromaggregat **********************************************************************************************************************************************************************

	//Eingänge
	Aktoren.Notstromaggregat.BetriebsmldgNotstromaggregat	:= diNotstromaggregatInBetrieb;

	//GUI-Parameter
	Aktoren.Notstromaggregat.Freigabe						:= Betriebsparameter.Ausstattung.Notstromaggregat;
	Aktoren.Notstromaggregat.QuitFehler						:= hmiButtons.QuitFehler;
	Aktoren.Notstromaggregat.VerzBetriebsmeldung			:= Betriebsparameter.Notstromaggregat.VerzBetriebsmeldung;
	Aktoren.Notstromaggregat.Vorlaufzeit					:= Betriebsparameter.Notstromaggregat.Vorlaufzeit;
	Aktoren.Notstromaggregat.Nachlaufzeit					:= Betriebsparameter.Notstromaggregat.Nachlaufzeit;

	//Ausgänge
	doNotstromaggregatEin									:= Aktoren.Notstromaggregat.FreigabeNotstromaggregatOut;

	//Status
	IF Aktoren.Notstromaggregat.NotstromBereitOut THEN
		gStatusAnlage.Aktor[AKTOR_NOTSTROMAGGREGAT]		:= STATUS_BEREIT;
	ELSIF doNotstromaggregatEin THEN
		gStatusAnlage.Aktor[AKTOR_NOTSTROMAGGREGAT]		:= STATUS_AKTIV;
	ELSIF Aktoren.Notstromaggregat.FehlerOut THEN
		gStatusAnlage.Aktor[AKTOR_NOTSTROMAGGREGAT]		:= STATUS_STOERUNG;
	ELSE
		gStatusAnlage.Aktor[AKTOR_NOTSTROMAGGREGAT]		:= STATUS_NICHT_AKTIV;
	END_IF

	//Brandschutzklappe **********************************************************************************************************************************************************************

	//Eingänge
	Aktoren.Brandschutzklappe.EndlageOffen					:= FALSE;
	Aktoren.Brandschutzklappe.EndlageGeschl					:= FALSE;
	Aktoren.Brandschutzklappe.LaufzeitOeffnen				:= 0;
	Aktoren.Brandschutzklappe.LaufzeitSchliessen			:= 0;
	Aktoren.Brandschutzklappe.Stoerung						:= FALSE;

	//GUI-Parameter
	Aktoren.Brandschutzklappe.QuitFehler					:= hmiButtons.QuitFehler;

	//Ausgänge
	doBrandschutzklappeAuf									:= Aktoren.Brandschutzklappe.OeffnenOut;

	//Status
	IF Aktoren.Brandschutzklappe.OeffnenOut THEN
		gStatusAnlage.Aktor[AKTOR_BRANDSCHUTZKLAPPE]	:= STATUS_OFFEN;
	ELSIF Betriebsparameter.Ausstattung.Brandschutzklappe THEN
		gStatusAnlage.Aktor[AKTOR_BRANDSCHUTZKLAPPE]	:= STATUS_GESCHLOSSEN;
	ELSE
		gStatusAnlage.Aktor[AKTOR_BRANDSCHUTZKLAPPE]	:= STATUS_NICHT_VERFUEGBAR;
	END_IF

END_PROGRAM
```

### Program Logical/IO/io407

#### Main.st
```iecst
PROGRAM _INIT

	hmiStatus.NameSteuerung	:= 0; //= LaTronic CControl 4.07

END_PROGRAM

PROGRAM _CYCLIC

	//Bei Konfiguration 4.07 -> Text auf Login-Seite anpassen, Option Entfeuchter ausschalten

	hmiParameter.Ausstattung.Entfeuchter := FALSE;
	hmiParameter.Ausstattung.Bypassklappe := FALSE;
	hmiParameter.Ausstattung.Box5 := FALSE;
	hmiParameter.Ausstattung.Box6 := FALSE;

	IF hmiParameter.Ausstattung.Abluftklappe THEN
		hmiParameter.Ausstattung.Abluftventilator := FALSE;
	ELSIF hmiParameter.Ausstattung.Abluftventilator THEN
		hmiParameter.Ausstattung.Abluftklappe := FALSE;
	END_IF

	//Zeitticks generieren
	fbLascoZdxx_0(IN 	:= Echtzeit.Sekunde);
	sekTick				:= fbLascoZdxx_0.Q;

	//=========================================================================================================================================================
	//IO-Zuweisung LaTronic CControl 4.07
	//=========================================================================================================================================================

	//Kein Testbetrieb
	IF (gAktModus <> IOTEST) THEN

		//MODUL 01 - BR7300 Busempfänger **********************************************************************************************************************
		brModul01;

		//MODUL 02 - CM8281 ***********************************************************************************************************************************
		//*****************************************************************************************************************************************************
		diVentilator1InBetrieb	:= cmModul02.di01;
		di24VDCinternIstOk		:= cmModul02.di02;
		//Reserve				:= cmModul02.di03;
		//Reserve				:= cmModul02.di04;

		cmModul02.do01			:= doVentilator1Ein;
		cmModul02.do02			:= doTrocknungInBetrieb;

		//Eingangssignale filtern
		IF sekTick THEN
			LCRMovAvgFlt_0(enable := TRUE, x := cmModul02.ai01, base := Betriebsparameter.Sensoren.FilterzeitFrischluft);
		END_IF

		//Frischluft Temperatur
		LCRLimScal_0(x := LCRMovAvgFlt_0.y, x1 := 0, y1 := Betriebsparameter.Sensoren.FrischlTempMessberMin,
		x2 := 32767, y2 := Betriebsparameter.Sensoren.FrischlTempMessberMax);
		aiFrischluftTemperatur		:= LCRLimScal_0.y + Betriebsparameter.Sensoren.OffsetFrischluftTemp;

		//Drehzahlvorgabe FU Ventilator 1
		LCRLimScal_0(x := aoDrehzahlvorgVentilator1, x1 := Betriebsparameter.Ventilator1.DrehzahlMin, y1 := 0,
		x2 := Betriebsparameter.Ventilator1.DrehzahlMax, y2 := 32767);
		cmModul02.ao01				:= REAL_TO_INT(LCRLimScal_0.y);

		//MODUL 03 - CM8281 ***********************************************************************************************************************************
		//*****************************************************************************************************************************************************
		diBox1Offen				:= cmModul03.di01;
		diBox1Geschl			:= cmModul03.di02;
		diBox2Offen				:= cmModul03.di03;
		diBox2Geschl			:= cmModul03.di04;

		cmModul03.do01			:= doFreigabeBox1;
		cmModul03.do02			:= doFreigabeBox2;

		//Eingangssignale filtern
		IF sekTick THEN
			LCRMovAvgFlt_1(enable := TRUE, x := cmModul03.ai01, base := Betriebsparameter.Sensoren.FilterzeitFrischluft);
		END_IF

		//Frischluft rel. Feuchte
		LCRLimScal_0(x := LCRMovAvgFlt_1.y, x1 := 0, y1 := Betriebsparameter.Sensoren.FrischlFeuchteMessberMin,
		x2 := 32767, y2 := Betriebsparameter.Sensoren.FrischlFeuchteMessberMax);
		aiFrischluftFeuchte		:= LCRLimScal_0.y + Betriebsparameter.Sensoren.OffsetFrischluftFeuchte;

		//Temperaturvorgabe Warmluftofen
		LCRLimScal_0(x := aoTemperaturvorgWarmluftofen, x1 := 0, y1 := 0,
		x2 := 100, y2 := 32767);
		cmModul03.ao01				:= REAL_TO_INT(LCRLimScal_0.y);

		//MODUL 04 - CM8281 ***********************************************************************************************************************************
		//*****************************************************************************************************************************************************
		diVentilator2InBetrieb			:= cmModul04.di01;
		diDrehzahlbegrVentilator1		:= cmModul04.di02;
		diDrehzahlbegrVentilator2		:= cmModul04.di03;
		//Reserve						:= cmModul04.di04;

		cmModul04.do01					:= doTrocknungStoerung;
		cmModul04.do02					:= doVentilator2Ein;

		//Eingangssignale filtern
		IF sekTick THEN
			LCRMovAvgFlt_2(enable := TRUE, x := cmModul04.ai01, base := Betriebsparameter.Sensoren.FilterzeitTrockenluft);
		END_IF

		//Trockenluft Temperatur
		LCRLimScal_0(x := LCRMovAvgFlt_2.y, x1 := 0, y1 := Betriebsparameter.Sensoren.TrockenlTempMessberMin,
		x2 := 32767, y2 := Betriebsparameter.Sensoren.TrockenlTempMessberMax);
		aiTrockenluftTemperatur		:= LCRLimScal_0.y + Betriebsparameter.Sensoren.OffsetTrockenluftTemp;

		//Drehzahlvorgabe FU Ventilator 2
		LCRLimScal_0(x := aoDrehzahlvorgVentilator2, x1 := Betriebsparameter.Ventilator2.DrehzahlMin, y1 := 0,
		x2 := Betriebsparameter.Ventilator2.DrehzahlMax, y2 := 32767);
		cmModul04.ao01				:= REAL_TO_INT(LCRLimScal_0.y);

		//MODUL 05 - CM8281 ***********************************************************************************************************************************
		//*****************************************************************************************************************************************************
		diWarmluftofenInBetrieb		:= cmModul05.di01;
		diScheitholzofenInBetrieb	:= cmModul05.di02;
		//Reserve					:= cmModul05.di03;
		//Reserve					:= cmModul05.di04;

		cmModul05.do01				:= doWarmluftofenEin;
		cmModul05.do02				:= doHeizregisterEin;

		//Eingangssignale filtern
		IF sekTick THEN
			LCRMovAvgFlt_3(enable := TRUE, x := cmModul05.ai01, base := Betriebsparameter.Sensoren.FilterzeitTrockenluft);
		END_IF

		//Trockenluft rel. Feuchte
		LCRLimScal_0(x := LCRMovAvgFlt_3.y, x1 := 0, y1 := Betriebsparameter.Sensoren.TrockenlFeuchteMessberMin,
		x2 := 32767, y2 := Betriebsparameter.Sensoren.TrockenlFeuchteMessberMax);
		aiTrockenluftFeuchte		:= LCRLimScal_0.y + Betriebsparameter.Sensoren.OffsetTrockenluftFeuchte;

		//Leistungsvorgabe Heizregister
		LCRLimScal_0(x := aoLeistungsvorgHeizregister, x1 := 0.0, y1 := 0, x2 := 100.0, y2 := 32767);
		cmModul05.ao01				:= REAL_TO_INT(LCRLimScal_0.y);

		//MODUL 06 - CM8281 ***********************************************************************************************************************************
		//*****************************************************************************************************************************************************
		diBox3Offen				:= cmModul06.di01;
		diBox3Geschl			:= cmModul06.di02;
		diBox4Offen				:= cmModul06.di03;
		diBox4Geschl			:= cmModul06.di04;

		cmModul06.do01			:= doFreigabeBox3;
		cmModul06.do02			:= doFreigabeBox4;

		//Eingangssignale filtern
		IF sekTick THEN
			LCRMovAvgFlt_4(enable := TRUE, x := cmModul06.ai01, base := Betriebsparameter.Sensoren.FilterzeitAbluft);
		END_IF

		//Abluft Temperatur
		LCRLimScal_0(x := LCRMovAvgFlt_4.y, x1 := 0, y1 := Betriebsparameter.Sensoren.AbluftTempMessberMin,
		x2 := 32767, y2 := Betriebsparameter.Sensoren.AbluftTempMessberMax);
		aiAbluftTemperatur		:= LCRLimScal_0.y + Betriebsparameter.Sensoren.OffsetAbluftTemp;

		//Analogausgang
		cmModul06.ao01				:= 0;	//Reserve

		//MODUL 07 - CM8281 ***********************************************************************************************************************************
		//*****************************************************************************************************************************************************
		diBox5Offen				:= cmModul07.di01;
		diBox5Geschl			:= cmModul07.di02;
		diBox6Offen				:= cmModul07.di03;
		diBox6Geschl			:= cmModul07.di04;

		cmModul07.do01			:= doFreigabeBox5;
		cmModul07.do02			:= doFreigabeBox6;

		//Eingangssignale filtern
		IF sekTick THEN
			LCRMovAvgFlt_5(enable := TRUE, x := cmModul07.ai01, base := Betriebsparameter.Sensoren.FilterzeitAbluft);
		END_IF

		//Abluft rel. Feuchte
		LCRLimScal_0(x := LCRMovAvgFlt_5.y, x1 := 0, y1 := Betriebsparameter.Sensoren.AbluftFeuchteMessberMin,
		x2 := 32767, y2 := Betriebsparameter.Sensoren.AbluftFeuchteMessberMax);
		aiAbluftFeuchte		:= LCRLimScal_0.y + Betriebsparameter.Sensoren.OffsetAbluftFeuchte;

		//Analogausgang
		cmModul07.ao01				:= 0;	//Reserve

		//MODUL 08 - CM8281 ***********************************************************************************************************************************
		//*****************************************************************************************************************************************************
		diAbluftventInBetrieb	:= cmModul08.di01;
		//Reserve				:= cmModul08.di02;
		//Reserve				:= cmModul08.di03;
		//Reserve				:= cmModul08.di04;

		cmModul08.do01			:= doBrandschutzklappeAuf;
		cmModul08.do02			:= doAbluftventilatorEin;

		//Eingangssignale filtern
		IF sekTick THEN
			LCRMovAvgFlt_6(enable := TRUE, x := cmModul08.ai01, base := Betriebsparameter.Sensoren.FilterzeitDachluft);
		END_IF

		//Dachluft Temperatur
		LCRLimScal_0(x := LCRMovAvgFlt_6.y, x1 := 0, y1 := Betriebsparameter.Sensoren.DachTempMessberMin,
		x2 := 32767, y2 := Betriebsparameter.Sensoren.DachTempMessberMax);
		aiDachluftTemperatur		:= LCRLimScal_0.y + Betriebsparameter.Sensoren.OffsetDachTemp;

		//Drehzahlvorgabe Abluftventilator
		LCRLimScal_0(x := aoDrehzahlvorgAbluftventilator, x1 := Betriebsparameter.Abluftventilator.DrehzahlMin, y1 := 0,
		x2 := Betriebsparameter.Abluftventilator.DrehzahlMax, y2 := 32767);
		cmModul08.ao01				:= REAL_TO_INT(LCRLimScal_0.y);

		//MODUL 09 - CM8281 ***********************************************************************************************************************************
		//*****************************************************************************************************************************************************
		diAbluftklappeOffen		:= cmModul09.di01;
		diAbluftklappeGeschl	:= cmModul09.di02;
		//Reserve				:= cmModul09.di03;
		//Reserve				:= cmModul09.di04;

		cmModul09.do01			:= doAbluftklappeFreigabe;
		cmModul09.do02			:= FALSE;	//Reserve

		//Eingangssignale filtern
		IF sekTick THEN
			LCRMovAvgFlt_7(enable := TRUE, x := cmModul09.ai01, base := Betriebsparameter.Sensoren.FilterzeitDachluft);
		END_IF

		//Dachluft rel. Feuchte
		LCRLimScal_0(x := LCRMovAvgFlt_7.y, x1 := 0, y1 := Betriebsparameter.Sensoren.DachFeuchteMessberMin,
		x2 := 32767, y2 := Betriebsparameter.Sensoren.DachFeuchteMessberMax);
		aiDachluftFeuchte		:= LCRLimScal_0.y + Betriebsparameter.Sensoren.OffsetDachFeuchte;

		//Analogausgang
		cmModul09.ao01				:= 0;	//Reserve

		//MODUL 10 - CM8281 ***********************************************************************************************************************************
		//*****************************************************************************************************************************************************
		diUmschaltklappe1Offen		:= cmModul10.di01;
		diUmschaltklappe1Geschl		:= cmModul10.di02;
		diUmschaltklappe2Offen		:= cmModul10.di03;
		diUmschaltklappe2Geschl		:= cmModul10.di04;

		cmModul10.do01				:= doUmluftklappe1Freigabe;
		cmModul10.do02				:= doUmluftklappe2Freigabe;

		//Eingangssignale filtern
		IF sekTick THEN
			LCRMovAvgFlt_8(enable := TRUE, x := cmModul10.ai01, base := Betriebsparameter.Sensoren.FilterzeitLuftgeschwindigkeit);
		END_IF

		//Luftgeschwindigkeit
		LCRLimScal_0(x := LCRMovAvgFlt_8.y, x1 := 0, y1 := Betriebsparameter.Sensoren.LuftgeschwMessberMin,
		x2 := 32767, y2 := Betriebsparameter.Sensoren.LuftgeschwMessberMax);
		aiLuftgeschwindigkeit		:= LCRLimScal_0.y + Betriebsparameter.Sensoren.OffsetLuftgeschw;

		//Analogausgang
		cmModul10.ao01				:= 0;	//Reserve

		//MODUL 11 - CM8281 ***********************************************************************************************************************************
		//*****************************************************************************************************************************************************
		diNotstromaggregatInBetrieb		:= cmModul11.di01;
		//Reserve						:= cmModul11.di02;
		//Reserve						:= cmModul11.di03;
		//Reserve						:= cmModul11.di04;

		cmModul11.do01					:= doNotstromaggregatEin;
		cmModul11.do02					:= FALSE;	//Reserve

		//Eingangssignale filtern
		IF sekTick THEN
			LCRMovAvgFlt_9(enable := TRUE, x := cmModul11.ai01, base := Betriebsparameter.Sensoren.FilterzeitKanaldruck);
		END_IF

		//Differenzdruck
		LCRLimScal_0(x := LCRMovAvgFlt_9.y, x1 := 0, y1 := Betriebsparameter.Sensoren.KanaldruckMessberMin,
		x2 := 32767, y2 := Betriebsparameter.Sensoren.KanaldruckMessberMax);
		aiDifferenzdruck		:= LCRLimScal_0.y + Betriebsparameter.Sensoren.OffsetKanaldruck;

		//Analogausgang
		cmModul11.ao01				:= 0;	//Reserve

		//Modulstatus - Auswertung **********************************************************************************************************************************
		//***********************************************************************************************************************************************************

		//Modul 02 Frischluft Temperatur ****************************************************************************
		IF (cmModul02.StatusInput01.1 = FALSE AND cmModul02.StatusInput01.0 = TRUE) THEN
			diStatusFrischluftTempMin	:= TRUE;
		ELSE
			diStatusFrischluftTempMin	:= FALSE;
		END_IF
		IF (cmModul02.StatusInput01.1 = TRUE AND cmModul02.StatusInput01.0 = FALSE ) THEN
			diStatusFrischluftTempMax	 := TRUE;
		ELSE
			diStatusFrischluftTempMax	 := FALSE;
		END_IF

		//Modul 03 Frischluft rel. Feuchte ****************************************************************************
		IF (cmModul03.StatusInput01.1 = FALSE AND cmModul03.StatusInput01.0 = TRUE) THEN
			diStatusFrischluftFeuchteMin	:= TRUE;
		ELSE
			diStatusFrischluftFeuchteMin	:= FALSE;
		END_IF
		IF (cmModul03.StatusInput01.1 = TRUE AND cmModul03.StatusInput01.0 = FALSE ) THEN
			diStatusFrischluftFeuchteMax	 := TRUE;
		ELSE
			diStatusFrischluftFeuchteMax	 := FALSE;
		END_IF

		//Modul 04 Trockenluft Temperatur ****************************************************************************
		IF (cmModul04.StatusInput01.1 = FALSE AND cmModul04.StatusInput01.0 = TRUE) THEN
			diStatusTrockenluftTempMin	:= TRUE;
		ELSE
			diStatusTrockenluftTempMin	:= FALSE;
		END_IF
		IF (cmModul04.StatusInput01.1 = TRUE AND cmModul04.StatusInput01.0 = FALSE ) THEN
			diStatusTrockenluftTempMax	 := TRUE;
		ELSE
			diStatusTrockenluftTempMax	 := FALSE;
		END_IF

		//Modul 05 Trockenluft rel. Feuchte ****************************************************************************
		IF (cmModul05.StatusInput01.1 = FALSE AND cmModul05.StatusInput01.0 = TRUE) THEN
			diStatusTrockenluftFeuchteMin	:= TRUE;
		ELSE
			diStatusTrockenluftFeuchteMin	:= FALSE;
		END_IF
		IF (cmModul05.StatusInput01.1 = TRUE AND cmModul05.StatusInput01.0 = FALSE ) THEN
			diStatusTrockenluftFeuchteMax	 := TRUE;
		ELSE
			diStatusTrockenluftFeuchteMax	 := FALSE;
		END_IF

		//Modul 06 Abluft Temperatur ****************************************************************************
		IF (cmModul06.StatusInput01.1 = FALSE AND cmModul06.StatusInput01.0 = TRUE) THEN
			diStatusAbluftTempMin	:= TRUE;
		ELSE
			diStatusAbluftTempMin	:= FALSE;
		END_IF
		IF (cmModul06.StatusInput01.1 = TRUE AND cmModul06.StatusInput01.0 = FALSE ) THEN
			diStatusAbluftTempMax	 := TRUE;
		ELSE
			diStatusAbluftTempMax	 := FALSE;
		END_IF

		//Modul 07 Abluft rel. Feuchte ****************************************************************************
		IF (cmModul07.StatusInput01.1 = FALSE AND cmModul07.StatusInput01.0 = TRUE) THEN
			diStatusAbluftFeuchteMin	:= TRUE;
		ELSE
			diStatusAbluftFeuchteMin	:= FALSE;
		END_IF
		IF (cmModul07.StatusInput01.1 = TRUE AND cmModul07.StatusInput01.0 = FALSE ) THEN
			diStatusAbluftFeuchteMax	 := TRUE;
		ELSE
			diStatusAbluftFeuchteMax	 := FALSE;
		END_IF

		//Modul 08 Dachluft Temperatur ****************************************************************************
		IF (cmModul08.StatusInput01.1 = FALSE AND cmModul08.StatusInput01.0 = TRUE) THEN
			diStatusDachluftTempMin	:= TRUE;
		ELSE
			diStatusDachluftTempMin	:= FALSE;
		END_IF
		IF (cmModul08.StatusInput01.1 = TRUE AND cmModul08.StatusInput01.0 = FALSE ) THEN
			diStatusDachluftTempMax	 := TRUE;
		ELSE
			diStatusDachluftTempMax	 := FALSE;
		END_IF

		//Modul 09 Dachluft rel. Feuchte ****************************************************************************
		IF (cmModul09.StatusInput01.1 = FALSE AND cmModul09.StatusInput01.0 = TRUE) THEN
			diStatusDachluftFeuchteMin	:= TRUE;
		ELSE
			diStatusDachluftFeuchteMin	:= FALSE;
		END_IF
		IF (cmModul09.StatusInput01.1 = TRUE AND cmModul09.StatusInput01.0 = FALSE ) THEN
			diStatusDachluftFeuchteMax	 := TRUE;
		ELSE
			diStatusDachluftFeuchteMax	 := FALSE;
		END_IF

		//Modul 10 Luftgeschwindigkeit ****************************************************************************
		IF (cmModul10.StatusInput01.1 = FALSE AND cmModul10.StatusInput01.0 = TRUE) THEN
			diStatusLuftgeschwMin	:= TRUE;
		ELSE
			diStatusLuftgeschwMin	:= FALSE;
		END_IF
		IF (cmModul10.StatusInput01.1 = TRUE AND cmModul10.StatusInput01.0 = FALSE ) THEN
			diStatusLuftgeschwMax	:= TRUE;
		ELSE
			diStatusLuftgeschwMax	 := FALSE;
		END_IF
		IF ((cmModul10.StatusInput01.1 = TRUE AND cmModul10.StatusInput01.0 = TRUE) OR cmModul10.ai01 >= 32767) THEN
			diStatusLuftgeschwDrahtbruch := TRUE;
		ELSE
			diStatusLuftgeschwDrahtbruch := FALSE;
		END_IF

		//Modul 11 Differenzdruck ****************************************************************************
		IF (cmModul11.StatusInput01.1 = FALSE AND cmModul11.StatusInput01.0 = TRUE) THEN
			diStatusDifferenzdruckMin	:= TRUE;
		ELSE
			diStatusDifferenzdruckMin	:= FALSE;
		END_IF
		IF (cmModul11.StatusInput01.1 = TRUE AND cmModul11.StatusInput01.0 = FALSE ) THEN
			diStatusDifferenzdruckMax	 := TRUE;
		ELSE
			diStatusDifferenzdruckMax	 := FALSE;
		END_IF

		//Ausgänge Testbetrieb rücksetzen, wenn IO-Test nicht aktiv
		hmiIoTest.DigitalOut.doAbluftklappeFreigabe		:= FALSE;
		hmiIoTest.DigitalOut.doAbluftventilatorEin		:= FALSE;
		hmiIoTest.DigitalOut.doBrandschutzklappeAuf		:= FALSE;
		hmiIoTest.DigitalOut.doBypassklappeOeffnen		:= FALSE;
		hmiIoTest.DigitalOut.doFreigabeBox1				:= FALSE;
		hmiIoTest.DigitalOut.doFreigabeBox2				:= FALSE;
		hmiIoTest.DigitalOut.doFreigabeBox3				:= FALSE;
		hmiIoTest.DigitalOut.doFreigabeBox4				:= FALSE;
		hmiIoTest.DigitalOut.doFreigabeBox5				:= FALSE;
		hmiIoTest.DigitalOut.doFreigabeBox6				:= FALSE;
		hmiIoTest.DigitalOut.doHeizregisterEin			:= FALSE;
		hmiIoTest.DigitalOut.doKompressorEinModul1		:= FALSE;
		hmiIoTest.DigitalOut.doKompressorEinModul2		:= FALSE;
		hmiIoTest.DigitalOut.doMagnetventilEinModul1	:= FALSE;
		hmiIoTest.DigitalOut.doMagnetventilEinModul2	:= FALSE;
		hmiIoTest.DigitalOut.doNotstromaggregatEin		:= FALSE;
		hmiIoTest.DigitalOut.doOelsumpfheizungEinModul1	:= FALSE;
		hmiIoTest.DigitalOut.doOelsumpfheizungEinModul2	:= FALSE;
		hmiIoTest.DigitalOut.doTrocknungInBetrieb		:= FALSE;
		hmiIoTest.DigitalOut.doTrocknungStoerung		:= FALSE;
		hmiIoTest.DigitalOut.doUmluftklappe1Freigabe	:= FALSE;
		hmiIoTest.DigitalOut.doUmluftklappe2Freigabe	:= FALSE;
		hmiIoTest.DigitalOut.doVentilator1Ein			:= FALSE;
		hmiIoTest.DigitalOut.doVentilator2Ein			:= FALSE;
		hmiIoTest.DigitalOut.doWarmluftofenEin			:= FALSE;

		hmiIoTest.AnalogOut.aoDrehzahlvorgAbluftventilator	:= 0.0;
		hmiIoTest.AnalogOut.aoDrehzahlvorgKompressorModul1	:= 0.0;
		hmiIoTest.AnalogOut.aoDrehzahlvorgKompressorModul2	:= 0.0;
		hmiIoTest.AnalogOut.aoDrehzahlvorgVentilator1		:= 0.0;
		hmiIoTest.AnalogOut.aoDrehzahlvorgVentilator2		:= 0.0;
		hmiIoTest.AnalogOut.aoLeistungsvorgHeizregister		:= 0.0;
		hmiIoTest.AnalogOut.aoTemperaturvorgWarmluftofen	:= 0.0;

	//==============================================================================================================================================================================================================
	//Testbetrieb
	//==============================================================================================================================================================================================================
	ELSE

		//MODUL 01 - BR7300 Busempfänger **********************************************************************************************************************

		//MODUL 02 - CM8281 ***********************************************************************************************************************************
		//*****************************************************************************************************************************************************
		hmiIoTest.DigitalIn.diVentilator1InBetrieb	:= cmModul02.di01;
		hmiIoTest.DigitalIn.di24VDCinternIstOk		:= cmModul02.di02;
		//Reserve									:= cmModul02.di03;
		//Reserve									:= cmModul02.di04;

		cmModul02.do01			:= hmiIoTest.DigitalOut.doVentilator1Ein;
		cmModul02.do02			:= hmiIoTest.DigitalOut.doTrocknungInBetrieb;

		//Eingangssignale filtern
		IF sekTick THEN
			LCRMovAvgFlt_0(enable := TRUE, x := cmModul02.ai01, base := Betriebsparameter.Sensoren.FilterzeitFrischluft);
		END_IF

		//Frischluft Temperatur
		LCRLimScal_0(x := LCRMovAvgFlt_0.y, x1 := 0, y1 := Betriebsparameter.Sensoren.FrischlTempMessberMin,
		x2 := 32767, y2 := Betriebsparameter.Sensoren.FrischlTempMessberMax);
		hmiIoTest.AnalogIn.aiFrischluftTemperatur		:= LCRLimScal_0.y + Betriebsparameter.Sensoren.OffsetFrischluftTemp;

		//Drehzahlvorgabe FU Ventilator 1
		LCRLimScal_0(x := hmiIoTest.AnalogOut.aoDrehzahlvorgVentilator1, x1 := Betriebsparameter.Ventilator1.DrehzahlMin, y1 := 0,
		x2 := Betriebsparameter.Ventilator1.DrehzahlMax, y2 := 32767);
		cmModul02.ao01				:= REAL_TO_INT(LCRLimScal_0.y);

		//MODUL 03 - CM8281 ***********************************************************************************************************************************
		//*****************************************************************************************************************************************************
		hmiIoTest.DigitalIn.diBox1Offen				:= cmModul03.di01;
		hmiIoTest.DigitalIn.diBox1Geschl			:= cmModul03.di02;
		hmiIoTest.DigitalIn.diBox2Offen				:= cmModul03.di03;
		hmiIoTest.DigitalIn.diBox2Geschl			:= cmModul03.di04;

		cmModul03.do01			:= hmiIoTest.DigitalOut.doFreigabeBox1;
		cmModul03.do02			:= hmiIoTest.DigitalOut.doFreigabeBox2;

		//Eingangssignale filtern
		IF sekTick THEN
			LCRMovAvgFlt_1(enable := TRUE, x := cmModul03.ai01, base := Betriebsparameter.Sensoren.FilterzeitFrischluft);
		END_IF

		//Frischluft rel. Feuchte
		LCRLimScal_0(x := LCRMovAvgFlt_1.y, x1 := 0, y1 := Betriebsparameter.Sensoren.FrischlFeuchteMessberMin,
		x2 := 32767, y2 := Betriebsparameter.Sensoren.FrischlFeuchteMessberMax);
		hmiIoTest.AnalogIn.aiFrischluftFeuchte		:= LCRLimScal_0.y + Betriebsparameter.Sensoren.OffsetFrischluftFeuchte;

		//Temperaturvorgabe Warmluftofen
		LCRLimScal_0(x := hmiIoTest.AnalogOut.aoTemperaturvorgWarmluftofen, x1 := 0, y1 := 0,
		x2 := 100, y2 := 32767);
		cmModul03.ao01				:= REAL_TO_INT(LCRLimScal_0.y);

		//MODUL 04 - CM8281 ***********************************************************************************************************************************
		//*****************************************************************************************************************************************************
		hmiIoTest.DigitalIn.diVentilator2InBetrieb			:= cmModul04.di01;
		hmiIoTest.DigitalIn.diDrehzahlbegrVentilator1		:= cmModul04.di02;
		hmiIoTest.DigitalIn.diDrehzahlbegrVentilator2		:= cmModul04.di03;
		//Reserve											:= cmModul04.di04;

		cmModul04.do01					:= hmiIoTest.DigitalOut.doTrocknungStoerung;
		cmModul04.do02					:= hmiIoTest.DigitalOut.doVentilator2Ein;

		//Eingangssignale filtern
		IF sekTick THEN
			LCRMovAvgFlt_2(enable := TRUE, x := cmModul04.ai01, base := Betriebsparameter.Sensoren.FilterzeitTrockenluft);
		END_IF

		//Trockenluft Temperatur
		LCRLimScal_0(x := LCRMovAvgFlt_2.y, x1 := 0, y1 := Betriebsparameter.Sensoren.TrockenlTempMessberMin,
		x2 := 32767, y2 := Betriebsparameter.Sensoren.TrockenlTempMessberMax);
		hmiIoTest.AnalogIn.aiTrockenluftTemperatur		:= LCRLimScal_0.y + Betriebsparameter.Sensoren.OffsetTrockenluftTemp;

		//Drehzahlvorgabe FU Ventilator 2
		LCRLimScal_0(x := hmiIoTest.AnalogOut.aoDrehzahlvorgVentilator2, x1 := Betriebsparameter.Ventilator2.DrehzahlMin, y1 := 0,
		x2 := Betriebsparameter.Ventilator2.DrehzahlMax, y2 := 32767);
		cmModul04.ao01				:= REAL_TO_INT(LCRLimScal_0.y);

		//MODUL 05 - CM8281 ***********************************************************************************************************************************
		//*****************************************************************************************************************************************************
		hmiIoTest.DigitalIn.diWarmluftofenInBetrieb		:= cmModul05.di01;
		hmiIoTest.DigitalIn.diScheitholzofenInBetrieb	:= cmModul05.di02;
		//Reserve										:= cmModul05.di03;
		//Reserve										:= cmModul05.di04;

		cmModul05.do01				:= hmiIoTest.DigitalOut.doWarmluftofenEin;
		cmModul05.do02				:= hmiIoTest.DigitalOut.doHeizregisterEin;

		//Eingangssignale filtern
		IF sekTick THEN
			LCRMovAvgFlt_3(enable := TRUE, x := cmModul05.ai01, base := Betriebsparameter.Sensoren.FilterzeitTrockenluft);
		END_IF

		//Trockenluft rel. Feuchte
		LCRLimScal_0(x := LCRMovAvgFlt_3.y, x1 := 0, y1 := Betriebsparameter.Sensoren.TrockenlFeuchteMessberMin,
		x2 := 32767, y2 := Betriebsparameter.Sensoren.TrockenlFeuchteMessberMax);
		hmiIoTest.AnalogIn.aiTrockenluftFeuchte		:= LCRLimScal_0.y + Betriebsparameter.Sensoren.OffsetTrockenluftFeuchte;

		//Leistungsvorgabe Heizregister
		LCRLimScal_0(x := hmiIoTest.AnalogOut.aoLeistungsvorgHeizregister, x1 := 0.0, y1 := 0, x2 := 100.0, y2 := 32767);
		cmModul05.ao01				:= REAL_TO_INT(LCRLimScal_0.y);

		//MODUL 06 - CM8281 ***********************************************************************************************************************************
		//*****************************************************************************************************************************************************
		hmiIoTest.DigitalIn.diBox3Offen				:= cmModul06.di01;
		hmiIoTest.DigitalIn.diBox3Geschl			:= cmModul06.di02;
		hmiIoTest.DigitalIn.diBox4Offen				:= cmModul06.di03;
		hmiIoTest.DigitalIn.diBox4Geschl			:= cmModul06.di04;

		cmModul06.do01			:= hmiIoTest.DigitalOut.doFreigabeBox3;
		cmModul06.do02			:= hmiIoTest.DigitalOut.doFreigabeBox4;

		//Eingangssignale filtern
		IF sekTick THEN
			LCRMovAvgFlt_4(enable := TRUE, x := cmModul06.ai01, base := Betriebsparameter.Sensoren.FilterzeitAbluft);
		END_IF

		//Abluft Temperatur
		LCRLimScal_0(x := LCRMovAvgFlt_4.y, x1 := 0, y1 := Betriebsparameter.Sensoren.AbluftTempMessberMin,
		x2 := 32767, y2 := Betriebsparameter.Sensoren.AbluftTempMessberMax);
		hmiIoTest.AnalogIn.aiAbluftTemperatur		:= LCRLimScal_0.y + Betriebsparameter.Sensoren.OffsetAbluftTemp;

		//Analogausgang
		cmModul06.ao01				:= 0;	//Reserve

		//MODUL 07 - CM8281 ***********************************************************************************************************************************
		//*****************************************************************************************************************************************************
		hmiIoTest.DigitalIn.diBox5Offen				:= cmModul07.di01;
		hmiIoTest.DigitalIn.diBox5Geschl			:= cmModul07.di02;
		hmiIoTest.DigitalIn.diBox6Offen				:= cmModul07.di03;
		hmiIoTest.DigitalIn.diBox6Geschl			:= cmModul07.di04;

		cmModul07.do01			:= hmiIoTest.DigitalOut.doFreigabeBox5;
		cmModul07.do02			:= hmiIoTest.DigitalOut.doFreigabeBox6;

		//Eingangssignale filtern
		IF sekTick THEN
			LCRMovAvgFlt_5(enable := TRUE, x := cmModul07.ai01, base := Betriebsparameter.Sensoren.FilterzeitAbluft);
		END_IF

		//Abluft rel. Feuchte
		LCRLimScal_0(x := LCRMovAvgFlt_5.y, x1 := 0, y1 := Betriebsparameter.Sensoren.AbluftFeuchteMessberMin,
		x2 := 32767, y2 := Betriebsparameter.Sensoren.AbluftFeuchteMessberMax);
		hmiIoTest.AnalogIn.aiAbluftFeuchte		:= LCRLimScal_0.y + Betriebsparameter.Sensoren.OffsetAbluftFeuchte;

		//Analogausgang
		cmModul07.ao01				:= 0;	//Reserve

		//MODUL 08 - CM8281 ***********************************************************************************************************************************
		//*****************************************************************************************************************************************************
		hmiIoTest.DigitalIn.diAbluftventInBetrieb	:= cmModul08.di01;
		//Reserve									:= cmModul08.di02;
		//Reserve									:= cmModul08.di03;
		//Reserve									:= cmModul08.di04;

		cmModul08.do01			:= hmiIoTest.DigitalOut.doBrandschutzklappeAuf;
		cmModul08.do02			:= hmiIoTest.DigitalOut.doAbluftventilatorEin;

		//Eingangssignale filtern
		IF sekTick THEN
			LCRMovAvgFlt_6(enable := TRUE, x := cmModul08.ai01, base := Betriebsparameter.Sensoren.FilterzeitDachluft);
		END_IF

		//Dachluft Temperatur
		LCRLimScal_0(x := LCRMovAvgFlt_6.y, x1 := 0, y1 := Betriebsparameter.Sensoren.DachTempMessberMin,
		x2 := 32767, y2 := Betriebsparameter.Sensoren.DachTempMessberMax);
		hmiIoTest.AnalogIn.aiDachluftTemperatur		:= LCRLimScal_0.y + Betriebsparameter.Sensoren.OffsetDachTemp;

		//Drehzahlvorgabe Abluftventilator
		LCRLimScal_0(x := hmiIoTest.AnalogOut.aoDrehzahlvorgAbluftventilator, x1 := Betriebsparameter.Abluftventilator.DrehzahlMin, y1 := 0,
		x2 := Betriebsparameter.Abluftventilator.DrehzahlMax, y2 := 32767);
		cmModul08.ao01				:= REAL_TO_INT(LCRLimScal_0.y);

		//MODUL 09 - CM8281 ***********************************************************************************************************************************
		//*****************************************************************************************************************************************************
		hmiIoTest.DigitalIn.diAbluftklappeOffen		:= cmModul09.di01;
		hmiIoTest.DigitalIn.diAbluftklappeGeschl	:= cmModul09.di02;
		//Reserve									:= cmModul09.di03;
		//Reserve									:= cmModul09.di04;

		cmModul09.do01			:= hmiIoTest.DigitalOut.doAbluftklappeFreigabe;
		cmModul09.do02			:= FALSE;	//Reserve

		//Eingangssignale filtern
		IF sekTick THEN
			LCRMovAvgFlt_7(enable := TRUE, x := cmModul09.ai01, base := Betriebsparameter.Sensoren.FilterzeitDachluft);
		END_IF

		//Dachluft rel. Feuchte
		LCRLimScal_0(x := LCRMovAvgFlt_7.y, x1 := 0, y1 := Betriebsparameter.Sensoren.DachFeuchteMessberMin,
		x2 := 32767, y2 := Betriebsparameter.Sensoren.DachFeuchteMessberMax);
		hmiIoTest.AnalogIn.aiDachluftFeuchte		:= LCRLimScal_0.y + Betriebsparameter.Sensoren.OffsetDachFeuchte;

		//Analogausgang
		cmModul09.ao01				:= 0;	//Reserve

		//MODUL 10 - CM8281 ***********************************************************************************************************************************
		//*****************************************************************************************************************************************************
		hmiIoTest.DigitalIn.diUmschaltklappe1Offen		:= cmModul10.di01;
		hmiIoTest.DigitalIn.diUmschaltklappe1Geschl		:= cmModul10.di02;
		hmiIoTest.DigitalIn.diUmschaltklappe2Offen		:= cmModul10.di03;
		hmiIoTest.DigitalIn.diUmschaltklappe2Geschl		:= cmModul10.di04;

		cmModul10.do01				:= hmiIoTest.DigitalOut.doUmluftklappe1Freigabe;
		cmModul10.do02				:= hmiIoTest.DigitalOut.doUmluftklappe2Freigabe;

		//Eingangssignale filtern
		IF sekTick THEN
			LCRMovAvgFlt_8(enable := TRUE, x := cmModul10.ai01, base := Betriebsparameter.Sensoren.FilterzeitLuftgeschwindigkeit);
		END_IF

		//Luftgeschwindigkeit
		LCRLimScal_0(x := LCRMovAvgFlt_8.y, x1 := 0, y1 := Betriebsparameter.Sensoren.LuftgeschwMessberMin,
		x2 := 32767, y2 := Betriebsparameter.Sensoren.LuftgeschwMessberMax);
		hmiIoTest.AnalogIn.aiLuftgeschwindigkeit		:= LCRLimScal_0.y + Betriebsparameter.Sensoren.OffsetLuftgeschw;

		//Analogausgang
		cmModul10.ao01				:= 0;	//Reserve

		//MODUL 11 - CM8281 ***********************************************************************************************************************************
		//*****************************************************************************************************************************************************
		hmiIoTest.DigitalIn.diNotstromaggregatInBetrieb		:= cmModul11.di01;
		//Reserve											:= cmModul11.di02;
		//Reserve											:= cmModul11.di03;
		//Reserve											:= cmModul11.di04;

		cmModul11.do01					:= hmiIoTest.DigitalOut.doNotstromaggregatEin;
		cmModul11.do02					:= FALSE;	//Reserve

		//Eingangssignale filtern
		IF sekTick THEN
			LCRMovAvgFlt_9(enable := TRUE, x := cmModul11.ai01, base := Betriebsparameter.Sensoren.FilterzeitKanaldruck);
		END_IF

		//Differenzdruck
		LCRLimScal_0(x := LCRMovAvgFlt_9.y, x1 := 0, y1 := Betriebsparameter.Sensoren.KanaldruckMessberMin,
		x2 := 32767, y2 := Betriebsparameter.Sensoren.KanaldruckMessberMax);
		hmiIoTest.AnalogIn.aiDifferenzdruck		:= LCRLimScal_0.y + Betriebsparameter.Sensoren.OffsetKanaldruck;

		//Analogausgang
		cmModul11.ao01				:= 0;	//Reserve

		//Modulstatus - Auswertung **********************************************************************************************************************************
		//***********************************************************************************************************************************************************

		//Modul 02 Frischluft Temperatur ****************************************************************************
		IF (cmModul02.StatusInput01.1 = FALSE AND cmModul02.StatusInput01.0 = TRUE) THEN
			hmiIoTest.StatusIn.diStatusFrischluftTempMin	:= TRUE;
		ELSE
			diStatusFrischluftTempMin	:= FALSE;
		END_IF
		IF (cmModul02.StatusInput01.1 = TRUE AND cmModul02.StatusInput01.0 = FALSE ) THEN
			hmiIoTest.StatusIn.diStatusFrischluftTempMax	 := TRUE;
		ELSE
			hmiIoTest.StatusIn.diStatusFrischluftTempMax	 := FALSE;
		END_IF

		//Modul 03 Frischluft rel. Feuchte ****************************************************************************
		IF (cmModul03.StatusInput01.1 = FALSE AND cmModul03.StatusInput01.0 = TRUE) THEN
			hmiIoTest.StatusIn.diStatusFrischluftFeuchteMin	:= TRUE;
		ELSE
			hmiIoTest.StatusIn.diStatusFrischluftFeuchteMin	:= FALSE;
		END_IF
		IF (cmModul03.StatusInput01.1 = TRUE AND cmModul03.StatusInput01.0 = FALSE ) THEN
			hmiIoTest.StatusIn.diStatusFrischluftFeuchteMax	 := TRUE;
		ELSE
			hmiIoTest.StatusIn.diStatusFrischluftFeuchteMax	 := FALSE;
		END_IF

		//Modul 04 Trockenluft Temperatur ****************************************************************************
		IF (cmModul04.StatusInput01.1 = FALSE AND cmModul04.StatusInput01.0 = TRUE) THEN
			hmiIoTest.StatusIn.diStatusTrockenluftTempMin	:= TRUE;
		ELSE
			hmiIoTest.StatusIn.diStatusTrockenluftTempMin	:= FALSE;
		END_IF
		IF (cmModul04.StatusInput01.1 = TRUE AND cmModul04.StatusInput01.0 = FALSE ) THEN
			hmiIoTest.StatusIn.diStatusTrockenluftTempMax	 := TRUE;
		ELSE
			hmiIoTest.StatusIn.diStatusTrockenluftTempMax	 := FALSE;
		END_IF

		//Modul 05 Trockenluft rel. Feuchte ****************************************************************************
		IF (cmModul05.StatusInput01.1 = FALSE AND cmModul05.StatusInput01.0 = TRUE) THEN
			hmiIoTest.StatusIn.diStatusTrockenluftFeuchteMin	:= TRUE;
		ELSE
			hmiIoTest.StatusIn.diStatusTrockenluftFeuchteMin	:= FALSE;
		END_IF
		IF (cmModul05.StatusInput01.1 = TRUE AND cmModul05.StatusInput01.0 = FALSE ) THEN
			hmiIoTest.StatusIn.diStatusTrockenluftFeuchteMax	 := TRUE;
		ELSE
			hmiIoTest.StatusIn.diStatusTrockenluftFeuchteMax	 := FALSE;
		END_IF

		//Modul 06 Abluft Temperatur ****************************************************************************
		IF (cmModul06.StatusInput01.1 = FALSE AND cmModul06.StatusInput01.0 = TRUE) THEN
			hmiIoTest.StatusIn.diStatusAbluftTempMin	:= TRUE;
		ELSE
			hmiIoTest.StatusIn.diStatusAbluftTempMin	:= FALSE;
		END_IF
		IF (cmModul06.StatusInput01.1 = TRUE AND cmModul06.StatusInput01.0 = FALSE ) THEN
			hmiIoTest.StatusIn.diStatusAbluftTempMax	 := TRUE;
		ELSE
			hmiIoTest.StatusIn.diStatusAbluftTempMax	 := FALSE;
		END_IF

		//Modul 07 Abluft rel. Feuchte ****************************************************************************
		IF (cmModul07.StatusInput01.1 = FALSE AND cmModul07.StatusInput01.0 = TRUE) THEN
			hmiIoTest.StatusIn.diStatusAbluftFeuchteMin	:= TRUE;
		ELSE
			hmiIoTest.StatusIn.diStatusAbluftFeuchteMin	:= FALSE;
		END_IF
		IF (cmModul07.StatusInput01.1 = TRUE AND cmModul07.StatusInput01.0 = FALSE ) THEN
			hmiIoTest.StatusIn.diStatusAbluftFeuchteMax	 := TRUE;
		ELSE
			hmiIoTest.StatusIn.diStatusAbluftFeuchteMax	 := FALSE;
		END_IF

		//Modul 08 Dachluft Temperatur ****************************************************************************
		IF (cmModul08.StatusInput01.1 = FALSE AND cmModul08.StatusInput01.0 = TRUE) THEN
			hmiIoTest.StatusIn.diStatusDachluftTempMin	:= TRUE;
		ELSE
			hmiIoTest.StatusIn.diStatusDachluftTempMin	:= FALSE;
		END_IF
		IF (cmModul08.StatusInput01.1 = TRUE AND cmModul08.StatusInput01.0 = FALSE ) THEN
			hmiIoTest.StatusIn.diStatusDachluftTempMax	 := TRUE;
		ELSE
			hmiIoTest.StatusIn.diStatusDachluftTempMax	 := FALSE;
		END_IF

		//Modul 09 Dachluft rel. Feuchte ****************************************************************************
		IF (cmModul09.StatusInput01.1 = FALSE AND cmModul09.StatusInput01.0 = TRUE) THEN
			hmiIoTest.StatusIn.diStatusDachluftFeuchteMin	:= TRUE;
		ELSE
			hmiIoTest.StatusIn.diStatusDachluftFeuchteMin	:= FALSE;
		END_IF
		IF (cmModul09.StatusInput01.1 = TRUE AND cmModul09.StatusInput01.0 = FALSE ) THEN
			hmiIoTest.StatusIn.diStatusDachluftFeuchteMax	 := TRUE;
		ELSE
			hmiIoTest.StatusIn.diStatusDachluftFeuchteMax	 := FALSE;
		END_IF

		//Modul 10 Luftgeschwindigkeit ****************************************************************************
		IF (cmModul10.StatusInput01.1 = FALSE AND cmModul10.StatusInput01.0 = TRUE) THEN
			hmiIoTest.StatusIn.diStatusLuftgeschwMin	:= TRUE;
		ELSE
			hmiIoTest.StatusIn.diStatusLuftgeschwMin	:= FALSE;
		END_IF
		IF (cmModul10.StatusInput01.1 = TRUE AND cmModul10.StatusInput01.0 = FALSE ) THEN
			hmiIoTest.StatusIn.diStatusLuftgeschwMax	:= TRUE;
		ELSE
			hmiIoTest.StatusIn.diStatusLuftgeschwMax	 := FALSE;
		END_IF
		IF ((cmModul10.StatusInput01.1 = TRUE AND cmModul10.StatusInput01.0 = TRUE) OR cmModul10.ai01 >= 32767) THEN
			hmiIoTest.StatusIn.diStatusLuftgeschwDrahtbruch := TRUE;
		ELSE
			hmiIoTest.StatusIn.diStatusLuftgeschwDrahtbruch := FALSE;
		END_IF

		//Modul 11 Differenzdruck ****************************************************************************
		IF (cmModul11.StatusInput01.1 = FALSE AND cmModul11.StatusInput01.0 = TRUE) THEN
			hmiIoTest.StatusIn.diStatusDifferenzdruckMin	:= TRUE;
		ELSE
			hmiIoTest.StatusIn.diStatusDifferenzdruckMin	:= FALSE;
		END_IF
		IF (cmModul11.StatusInput01.1 = TRUE AND cmModul11.StatusInput01.0 = FALSE ) THEN
			hmiIoTest.StatusIn.diStatusDifferenzdruckMax	 := TRUE;
		ELSE
			hmiIoTest.StatusIn.diStatusDifferenzdruckMax	 := FALSE;
		END_IF

	END_IF

	//============================================================================================================================================================================
	//Modulüberwachungen
	//============================================================================================================================================================================

	loc_Erforderl_Mod1	:= TRUE;
	loc_Erforderl_Mod2	:= TRUE;
	loc_Erforderl_Mod3	:= Aktoren.VentUndKlappen.Boxenklappe1Vorhanden OR Aktoren.VentUndKlappen.Boxenklappe2Vorhanden OR
		Betriebsparameter.Ausstattung.SensorFrischluft OR Betriebsparameter.Ausstattung.WarmluftofenTempVorgabe;
	loc_Erforderl_Mod4	:= TRUE;
	loc_Erforderl_Mod5	:= Betriebsparameter.Ausstattung.Warmluftofen OR Betriebsparameter.Ausstattung.Scheitholzofen OR Betriebsparameter.Ausstattung.Heizregister OR
		Betriebsparameter.Ausstattung.SensorTrockenluft;
	loc_Erforderl_Mod6	:= Aktoren.VentUndKlappen.Boxenklappe3Vorhanden OR Aktoren.VentUndKlappen.Boxenklappe4Vorhanden OR Betriebsparameter.Ausstattung.SensorAbluft;
	loc_Erforderl_Mod7	:= Betriebsparameter.Ausstattung.SensorAbluft;
	loc_Erforderl_Mod8	:= Betriebsparameter.Ausstattung.Abluftventilator OR Betriebsparameter.Ausstattung.Brandschutzklappe OR Betriebsparameter.Ausstattung.SensorDachluft;
	loc_Erforderl_Mod9	:= Betriebsparameter.Ausstattung.Abluftklappe OR Betriebsparameter.Ausstattung.SensorDachluft;
	loc_Erforderl_Mod10	:= Betriebsparameter.Ausstattung.Umschaltklappe1 OR Betriebsparameter.Ausstattung.Umschaltklappe2 OR
		Betriebsparameter.Ausstattung.SensorLuftgeschwindigkeit;
	loc_Erforderl_Mod11	:= Betriebsparameter.Ausstattung.Notstromaggregat OR Betriebsparameter.Ausstattung.SensorKanaldruck;
	loc_Erforderl_Mod12	:= Betriebsparameter.Ausstattung.Energiemessung;

	fbLascoFehl_0.FehlerIn	:= (loc_Erforderl_Mod1 AND NOT brModul01.ModulOk) OR (loc_Erforderl_Mod2 AND NOT cmModul02.ModulOk) OR
	(loc_Erforderl_Mod3 AND NOT cmModul03.ModulOk) OR (loc_Erforderl_Mod4 AND NOT cmModul04.ModulOk) OR (loc_Erforderl_Mod5 AND NOT cmModul05.ModulOk) OR
	(loc_Erforderl_Mod6 AND NOT cmModul06.ModulOk) OR (loc_Erforderl_Mod7 AND NOT cmModul07.ModulOk) OR (loc_Erforderl_Mod8 AND NOT cmModul08.ModulOk) OR
	(loc_Erforderl_Mod9 AND NOT cmModul09.ModulOk) OR (loc_Erforderl_Mod10 AND NOT cmModul10.ModulOk) OR (loc_Erforderl_Mod11 AND NOT cmModul11.ModulOk) OR
	(loc_Erforderl_Mod12 AND NOT gEnergiemessungModulOk);
	fbLascoFehl_0.Mode		:= 2;
	fbLascoFehl_0.Quit		:= hmiButtons.QuitFehler;
	fbLascoFehl_0.Tick		:= sekTick;
	fbLascoFehl_0();

	alarmSystem[FEHLER_KOMMUNIKATION_DISPLAY_IO] := fbLascoFehl_0.FehlerOut;

END_PROGRAM

PROGRAM _EXIT

END_PROGRAM
```

### Program Logical/Regelung/Leistung
